LIN {X 0,Y 349.295,Z 384.118,A -85,B 0,C 180,E1 -15532.689,E2 -15532.689} C_VEL
LIN {X 0,Y 344.629,Z 399.806,A -85,B 0,C 180,E1 -15533.924,E2 -15533.924} C_VEL
LIN {X 0,Y 339.086,Z 417.351,A -85,B 0,C 180,E1 -15535.611,E2 -15535.611} C_VEL
LIN {X 0,Y 333.971,Z 433.133,A -85,B 0,C 180,E1 -15537.457,E2 -15537.457} C_VEL
LIN {X 0,Y 329.124,Z 447.831,A -85,B 0,C 180,E1 -15539.525,E2 -15539.525} C_VEL
LIN {X 0,Y 324.634,Z 461.889,A -85,B 0,C 180,E1 -15541.909,E2 -15541.909} C_VEL
LIN {X 0,Y 320.374,Z 475.464,A -85,B 0,C 180,E1 -15544.673,E2 -15544.673} C_VEL
LIN {X 0,Y 317.065,Z 486.958,A -85,B 0,C 180,E1 -15547.519,E2 -15547.519} C_VEL
LIN {X 0,Y 314.518,Z 496.621,A -85,B 0,C 180,E1 -15550.416,E2 -15550.416} C_VEL
LIN {X 0,Y 312.895,Z 503.797,A -85,B 0,C 180,E1 -15553.022,E2 -15553.022} C_VEL
LIN {X 0,Y 311.835,Z 509.983,A -85,B 0,C 180,E1 -15555.722,E2 -15555.722} C_VEL
LIN {X 0,Y 311.142,Z 514.648,A -85,B 0,C 180,E1 -15558.27,E2 -15558.27} C_VEL
LIN {X 0,Y 310.892,Z 518.384,A -85,B 0,C 180,E1 -15560.894,E2 -15560.894} C_VEL
LIN {X 0,Y 310.985,Z 521.013,A -85,B 0,C 180,E1 -15563.511,E2 -15563.511} C_VEL
LIN {X 0,Y 310.999,Z 522.524,A -85,B 0,C 180,E1 -15566.112,E2 -15566.112} C_VEL
LIN {X 0,Y 311.174,Z 522.908,A -85,B 0,C 180,E1 -15567.41,E2 -15567.41} C_VEL
LIN {X 0,Y 311.35,Z 522.705,A -85,B 0,C 180,E1 -15569.999,E2 -15569.999} C_VEL
LIN {X 0,Y 311.281,Z 521.372,A -85,B 0,C 180,E1 -15572.587,E2 -15572.587} C_VEL
LIN {X 0,Y 311.146,Z 518.832,A -85,B 0,C 180,E1 -15575.183,E2 -15575.183} C_VEL
LIN {X 0,Y 311.178,Z 516.141,A -85,B 0,C 180,E1 -15577.134,E2 -15577.134} C_VEL
LIN {X 0,Y 311.09,Z 511.33,A -85,B 0,C 180,E1 -15579.754,E2 -15579.754} C_VEL
LIN {X 0,Y 311.378,Z 505.192,A -85,B 0,C 180,E1 -15582.381,E2 -15582.381} C_VEL
LIN {X 0,Y 311.923,Z 497.582,A -85,B 0,C 180,E1 -15585.016,E2 -15585.016} C_VEL
LIN {X 0,Y 312.908,Z 488.328,A -85,B 0,C 180,E1 -15587.65,E2 -15587.65} C_VEL
LIN {X 0,Y 314.056,Z 478.588,A -85,B 0,C 180,E1 -15589.969,E2 -15589.969} C_VEL
LIN {X 0,Y 315.698,Z 467.285,A -85,B 0,C 180,E1 -15592.237,E2 -15592.237} C_VEL
LIN {X 0,Y 317.471,Z 454.864,A -85,B 0,C 180,E1 -15594.349,E2 -15594.349} C_VEL
LIN {X 0,Y 319.434,Z 441.443,A -85,B 0,C 180,E1 -15596.28,E2 -15596.28} C_VEL
LIN {X 0,Y 321.67,Z 427.047,A -85,B 0,C 180,E1 -15598.017,E2 -15598.017} C_VEL
LIN {X 0,Y 323.604,Z 413.175,A -85,B 0,C 180,E1 -15599.429,E2 -15599.429} C_VEL
LIN {X 0,Y 325.822,Z 396.562,A -85,B 0,C 180,E1 -15600.815,E2 -15600.815} C_VEL
LIN {X 0,Y 327.852,Z 379.404,A -85,B 0,C 180,E1 -15601.951,E2 -15601.951} C_VEL
LIN {X 0,Y 329.659,Z 361.75,A -85,B 0,C 180,E1 -15602.839,E2 -15602.839} C_VEL
LIN {X 0,Y 330.906,Z 344.404,A -85,B 0,C 180,E1 -15603.472,E2 -15603.472} C_VEL
LIN {X 0,Y 339.444,Z 199.123,A -85,B 0,C 180,E1 -15607.77,E2 -15607.77} C_VEL
LIN {X 0,Y 337.215,Z 179.474,A -85,B 0,C 180,E1 -15608.653,E2 -15608.653} C_VEL
LIN {X 0,Y 322.802,Z 147.216,A -85,B 0,C 180,E1 -15611.25,E2 -15611.25} C_VEL
LIN {X 0,Y 320.937,Z 143.018,A -85,B 0,C 180,E1 -15611.632,E2 -15611.632} C_VEL
LIN {X 0,Y 315.137,Z 125.785,A -85,B 0,C 180,E1 -15614.923,E2 -15614.923} C_VEL
LIN {X 0,Y 312.533,Z 117.869,A -85,B 0,C 180,E1 -15616.557,E2 -15616.557} C_VEL
LIN {X 0,Y 312.504,Z 117.869,A -85,B 0,C 180,E1 -15620.972,E2 -15620.972} C_VEL
LIN {X 0,Y 312.528,Z 117.87,A -85,B 0,C 180,E1 -15624.22,E2 -15624.22} C_VEL
LIN {X 0,Y 312.503,Z 117.868,A -85,B 0,C 180,E1 -15627.334,E2 -15627.334} C_VEL
LIN {X 0,Y 312.548,Z 117.863,A -85,B 0,C 180,E1 -15631.276,E2 -15631.276} C_VEL
LIN {X 0,Y 312.581,Z 117.86,A -85,B 0,C 180,E1 -15634.711,E2 -15634.711} C_VEL
LIN {X 0,Y 312.582,Z 117.86,A -85,B 0,C 180,E1 -15637.529,E2 -15637.529} C_VEL
LIN {X 0,Y 312.634,Z 117.855,A -85,B 0,C 180,E1 -15641.656,E2 -15641.656} C_VEL
LIN {X 0,Y 312.69,Z 117.848,A -85,B 0,C 180,E1 -15645.686,E2 -15645.686} C_VEL
LIN {X 0,Y 312.699,Z 117.846,A -85,B 0,C 180,E1 -15649.642,E2 -15649.642} C_VEL
LIN {X 0,Y 312.867,Z 117.824,A -85,B 0,C 180,E1 -15652.254,E2 -15652.254} C_VEL
LIN {X 0,Y 312.714,Z 117.839,A -85,B 0,C 180,E1 -15654.842,E2 -15654.842} C_VEL
LIN {X 0,Y 312.986,Z 117.808,A -85,B 0,C 180,E1 -15658.713,E2 -15658.713} C_VEL
LIN {X 0,Y 313.116,Z 117.794,A -85,B 0,C 180,E1 -15660,E2 -15660} C_VEL
LIN {X 0,Y 312.934,Z 117.814,A -85,B 0,C 180,E1 -15662.575,E2 -15662.575} C_VEL
LIN {X 0,Y 312.89,Z 117.818,A -85,B 0,C 180,E1 -15666.639,E2 -15666.639} C_VEL
LIN {X 0,Y 312.783,Z 117.835,A -85,B 0,C 180,E1 -15669.049,E2 -15669.049} C_VEL
LIN {X 0,Y 312.63,Z 117.853,A -85,B 0,C 180,E1 -15672.991,E2 -15672.991} C_VEL
LIN {X 0,Y 312.634,Z 117.854,A -85,B 0,C 180,E1 -15675.65,E2 -15675.65} C_VEL
LIN {X 0,Y 312.626,Z 117.857,A -85,B 0,C 180,E1 -15679.237,E2 -15679.237} C_VEL
LIN {X 0,Y 312.542,Z 117.864,A -85,B 0,C 180,E1 -15682.79,E2 -15682.79} C_VEL
LIN {X 0,Y 312.592,Z 117.857,A -85,B 0,C 180,E1 -15685.934,E2 -15685.934} C_VEL
LIN {X 0,Y 312.534,Z 117.864,A -85,B 0,C 180,E1 -15689.651,E2 -15689.651} C_VEL
LIN {X 0,Y 312.515,Z 117.867,A -85,B 0,C 180,E1 -15693.689,E2 -15693.689} C_VEL
LIN {X 0,Y 312.517,Z 117.867,A -85,B 0,C 180,E1 -15697.386,E2 -15697.386} C_VEL
LIN {X 0,Y 312.486,Z 117.873,A -85,B 0,C 180,E1 -15700.71,E2 -15700.71} C_VEL
LIN {X 0,Y 312.472,Z 117.872,A -85,B 0,C 180,E1 -15704.206,E2 -15704.206} C_VEL
LIN {X 0,Y 312.529,Z 117.864,A -85,B 0,C 180,E1 -15707.91,E2 -15707.91} C_VEL
LIN {X 0,Y 312.54,Z 117.863,A -85,B 0,C 180,E1 -15711.909,E2 -15711.909} C_VEL
LIN {X 0,Y 312.504,Z 117.867,A -85,B 0,C 180,E1 -15715.791,E2 -15715.791} C_VEL
LIN {X 0,Y 312.518,Z 117.869,A -85,B 0,C 180,E1 -15718.854,E2 -15718.854} C_VEL
LIN {X 0,Y 312.568,Z 117.858,A -85,B 0,C 180,E1 -15721.825,E2 -15721.825} C_VEL
LIN {X 0,Y 312.584,Z 117.861,A -85,B 0,C 180,E1 -15724.712,E2 -15724.712} C_VEL
LIN {X 0,Y 312.587,Z 117.857,A -85,B 0,C 180,E1 -15727.53,E2 -15727.53} C_VEL
LIN {X 0,Y 312.638,Z 117.851,A -85,B 0,C 180,E1 -15731.657,E2 -15731.657} C_VEL
LIN {X 0,Y 312.693,Z 117.844,A -85,B 0,C 180,E1 -15735.687,E2 -15735.687} C_VEL
LIN {X 0,Y 312.702,Z 117.844,A -85,B 0,C 180,E1 -15739.643,E2 -15739.643} C_VEL
LIN {X 0,Y 312.872,Z 117.827,A -85,B 0,C 180,E1 -15742.255,E2 -15742.255} C_VEL
LIN {X 0,Y 312.718,Z 117.841,A -85,B 0,C 180,E1 -15744.843,E2 -15744.843} C_VEL
LIN {X 0,Y 312.989,Z 117.808,A -85,B 0,C 180,E1 -15748.714,E2 -15748.714} C_VEL
LIN {X 0,Y 312.989,Z 117.807,A -85,B 0,C 180,E1 -15751.288,E2 -15751.288} C_VEL
LIN {X 0,Y 312.718,Z 117.84,A -85,B 0,C 180,E1 -15755.158,E2 -15755.158} C_VEL
LIN {X 0,Y 312.873,Z 117.826,A -85,B 0,C 180,E1 -15757.747,E2 -15757.747} C_VEL
LIN {X 0,Y 312.671,Z 117.849,A -85,B 0,C 180,E1 -15761.672,E2 -15761.672} C_VEL
LIN {X 0,Y 312.702,Z 117.844,A -85,B 0,C 180,E1 -15764.888,E2 -15764.888} C_VEL
LIN {X 0,Y 312.632,Z 117.852,A -85,B 0,C 180,E1 -15769.237,E2 -15769.237} C_VEL
LIN {X 0,Y 312.548,Z 117.861,A -85,B 0,C 180,E1 -15772.79,E2 -15772.79} C_VEL
LIN {X 0,Y 312.605,Z 117.858,A -85,B 0,C 180,E1 -15775.936,E2 -15775.936} C_VEL
LIN {X 0,Y 312.54,Z 117.868,A -85,B 0,C 180,E1 -15779.651,E2 -15779.651} C_VEL
LIN {X 0,Y 312.522,Z 117.869,A -85,B 0,C 180,E1 -15783.689,E2 -15783.689} C_VEL
LIN {X 0,Y 312.541,Z 117.868,A -85,B 0,C 180,E1 -15787.384,E2 -15787.384} C_VEL
LIN {X 0,Y 312.493,Z 117.869,A -85,B 0,C 180,E1 -15790.71,E2 -15790.71} C_VEL
LIN {X 0,Y 312.476,Z 117.872,A -85,B 0,C 180,E1 -15794.206,E2 -15794.206} C_VEL
LIN {X 0,Y 312.489,Z 117.872,A -85,B 0,C 180,E1 -15797.919,E2 -15797.919} C_VEL
LIN {X 0,Y 312.489,Z 117.887,A -85,B 0,C 180,E1 -15798.632,E2 -15798.632} C_VEL
LIN {X 0,Y 313.513,Z 120.747,A -85,B 0,C 180,E1 -15798.857,E2 -15798.857} C_VEL
LIN {X 0,Y 325.494,Z 143.603,A -85,B 0,C 180,E1 -15800.977,E2 -15800.977} C_VEL
LIN {X 0,Y 338.412,Z 169.69,A -85,B 0,C 180,E1 -15803.121,E2 -15803.121} C_VEL
LIN {X 0,Y 336.711,Z 199.183,A -85,B 0,C 180,E1 -15803.99,E2 -15803.99} C_VEL
LIN {X 0,Y 331.473,Z 290.627,A -85,B 0,C 180,E1 -15806.67,E2 -15806.67} C_VEL
LIN {X 0,Y 330.453,Z 296.401,A -85,B 0,C 180,E1 -15806.798,E2 -15806.798} C_VEL
LIN {X 0,Y 323.959,Z 315.007,A -85,B 0,C 180,E1 -15807.144,E2 -15807.144} C_VEL
LIN {X 0,Y 322.988,Z 320.671,A -85,B 0,C 180,E1 -15807.384,E2 -15807.384} C_VEL
LIN {X 0,Y 321.504,Z 337.305,A -85,B 0,C 180,E1 -15808.356,E2 -15808.356} C_VEL
LIN {X 0,Y 319.895,Z 352.792,A -85,B 0,C 180,E1 -15809.495,E2 -15809.495} C_VEL
LIN {X 0,Y 318.015,Z 368.566,A -85,B 0,C 180,E1 -15810.909,E2 -15810.909} C_VEL
LIN {X 0,Y 315.817,Z 384.138,A -85,B 0,C 180,E1 -15812.592,E2 -15812.592} C_VEL
LIN {X 0,Y 313.777,Z 398.504,A -85,B 0,C 180,E1 -15814.459,E2 -15814.459} C_VEL
LIN {X 0,Y 311.835,Z 411.307,A -85,B 0,C 180,E1 -15816.419,E2 -15816.419} C_VEL
LIN {X 0,Y 309.955,Z 424.018,A -85,B 0,C 180,E1 -15818.728,E2 -15818.728} C_VEL
LIN {X 0,Y 308.326,Z 434.772,A -85,B 0,C 180,E1 -15821.046,E2 -15821.046} C_VEL
LIN {X 0,Y 307.039,Z 443.961,A -85,B 0,C 180,E1 -15823.374,E2 -15823.374} C_VEL
LIN {X 0,Y 305.92,Z 452.844,A -85,B 0,C 180,E1 -15826.041,E2 -15826.041} C_VEL
LIN {X 0,Y 305.072,Z 460.203,A -85,B 0,C 180,E1 -15828.707,E2 -15828.707} C_VEL
LIN {X 0,Y 304.599,Z 466.158,A -85,B 0,C 180,E1 -15831.374,E2 -15831.374} C_VEL
LIN {X 0,Y 304.269,Z 470.833,A -85,B 0,C 180,E1 -15834.034,E2 -15834.034} C_VEL
LIN {X 0,Y 304.16,Z 473.616,A -85,B 0,C 180,E1 -15836.025,E2 -15836.025} C_VEL
LIN {X 0,Y 304.172,Z 476.328,A -85,B 0,C 180,E1 -15838.676,E2 -15838.676} C_VEL
LIN {X 0,Y 304.288,Z 478.039,A -85,B 0,C 180,E1 -15841.323,E2 -15841.323} C_VEL
LIN {X 0,Y 304.671,Z 478.631,A -85,B 0,C 180,E1 -15843.968,E2 -15843.968} C_VEL
LIN {X 0,Y 305.028,Z 478.313,A -85,B 0,C 180,E1 -15846.615,E2 -15846.615} C_VEL
LIN {X 0,Y 305.938,Z 476.894,A -85,B 0,C 180,E1 -15849.253,E2 -15849.253} C_VEL
LIN {X 0,Y 307.056,Z 474.523,A -85,B 0,C 180,E1 -15851.888,E2 -15851.888} C_VEL
LIN {X 0,Y 308.567,Z 471.116,A -85,B 0,C 180,E1 -15854.509,E2 -15854.509} C_VEL
LIN {X 0,Y 310.423,Z 466.643,A -85,B 0,C 180,E1 -15857.117,E2 -15857.117} C_VEL
LIN {X 0,Y 312.955,Z 461.065,A -85,B 0,C 180,E1 -15859.685,E2 -15859.685} C_VEL
LIN {X 0,Y 315.894,Z 454.246,A -85,B 0,C 180,E1 -15862.223,E2 -15862.223} C_VEL
LIN {X 0,Y 319.439,Z 446.086,A -85,B 0,C 180,E1 -15864.709,E2 -15864.709} C_VEL
LIN {X 0,Y 323.477,Z 436.53,A -85,B 0,C 180,E1 -15867.145,E2 -15867.145} C_VEL
LIN {X 0,Y 328.04,Z 425.33,A -85,B 0,C 180,E1 -15869.522,E2 -15869.522} C_VEL
LIN {X 0,Y 333.3,Z 412.161,A -85,B 0,C 180,E1 -15871.813,E2 -15871.813} C_VEL
LIN {X 0,Y 338.512,Z 398.159,A -85,B 0,C 180,E1 -15873.853,E2 -15873.853} C_VEL
LIN {X 0,Y 343.392,Z 384.43,A -85,B 0,C 180,E1 -15875.502,E2 -15875.502} C_VEL
LIN {X 0,Y 348.987,Z 367.579,A -85,B 0,C 180,E1 -15877.167,E2 -15877.167} C_VEL
LIN {X 0,Y 354.438,Z 349.416,A -85,B 0,C 180,E1 -15878.611,E2 -15878.611} C_VEL
LIN {X 0,Y 358.655,Z 333.375,A -85,B 0,C 180,E1 -15879.625,E2 -15879.625} C_VEL
LIN {X 0,Y 362.306,Z 317.392,A -85,B 0,C 180,E1 -15880.415,E2 -15880.415} C_VEL
LIN {X 0,Y 369.736,Z 283.735,A -85,B 0,C 180,E1 -15881.704,E2 -15881.704} C_VEL
LIN {X 0,Y 385.229,Z 220.867,A -85,B 0,C 180,E1 -15883.972,E2 -15883.972} C_VEL
LIN {X 0,Y 386.116,Z 217.532,A -85,B 0,C 180,E1 -15884.081,E2 -15884.081} C_VEL
LIN {X 0,Y 385.94,Z 218.526,A -85,B 0,C 180,E1 -15884.797,E2 -15884.797} C_VEL
LIN {X 0,Y 369.925,Z 285.407,A -85,B 0,C 180,E1 -15887.172,E2 -15887.172} C_VEL
LIN {X 0,Y 357.945,Z 341.127,A -85,B 0,C 180,E1 -15889.289,E2 -15889.289} C_VEL
LIN {X 0,Y 352.257,Z 362.801,A -85,B 0,C 180,E1 -15890.323,E2 -15890.323} C_VEL
LIN {X 0,Y 346.181,Z 382.739,A -85,B 0,C 180,E1 -15891.556,E2 -15891.556} C_VEL
LIN {X 0,Y 341.651,Z 396.692,A -85,B 0,C 180,E1 -15892.638,E2 -15892.638} C_VEL
LIN {X 0,Y 335.68,Z 414.246,A -85,B 0,C 180,E1 -15894.294,E2 -15894.294} C_VEL
LIN {X 0,Y 330.21,Z 429.88,A -85,B 0,C 180,E1 -15896.104,E2 -15896.104} C_VEL
LIN {X 0,Y 325.165,Z 443.856,A -85,B 0,C 180,E1 -15898.025,E2 -15898.025} C_VEL
LIN {X 0,Y 320.164,Z 458.156,A -85,B 0,C 180,E1 -15900.402,E2 -15900.402} C_VEL
LIN {X 0,Y 315.91,Z 470.554,A -85,B 0,C 180,E1 -15902.857,E2 -15902.857} C_VEL
LIN {X 0,Y 312.361,Z 481.394,A -85,B 0,C 180,E1 -15905.402,E2 -15905.402} C_VEL
LIN {X 0,Y 309.46,Z 490.728,A -85,B 0,C 180,E1 -15907.992,E2 -15907.992} C_VEL
LIN {X 0,Y 307.28,Z 498.66,A -85,B 0,C 180,E1 -15910.631,E2 -15910.631} C_VEL
LIN {X 0,Y 305.658,Z 505.427,A -85,B 0,C 180,E1 -15913.296,E2 -15913.296} C_VEL
LIN {X 0,Y 304.618,Z 511.205,A -85,B 0,C 180,E1 -15916.109,E2 -15916.109} C_VEL
LIN {X 0,Y 304.111,Z 514.415,A -85,B 0,C 180,E1 -15917.995,E2 -15917.995} C_VEL
LIN {X 0,Y 303.814,Z 517.998,A -85,B 0,C 180,E1 -15920.68,E2 -15920.68} C_VEL
LIN {X 0,Y 303.901,Z 520.568,A -85,B 0,C 180,E1 -15923.359,E2 -15923.359} C_VEL
LIN {X 0,Y 303.924,Z 521.949,A -85,B 0,C 180,E1 -15926.021,E2 -15926.021} C_VEL
LIN {X 0,Y 304.173,Z 522.312,A -85,B 0,C 180,E1 -15928.675,E2 -15928.675} C_VEL
LIN {X 0,Y 304.296,Z 522.014,A -85,B 0,C 180,E1 -15929.999,E2 -15929.999} C_VEL
LIN {X 0,Y 304.222,Z 520.551,A -85,B 0,C 180,E1 -15932.647,E2 -15932.647} C_VEL
LIN {X 0,Y 304.095,Z 517.939,A -85,B 0,C 180,E1 -15935.303,E2 -15935.303} C_VEL
LIN {X 0,Y 304.12,Z 515.109,A -85,B 0,C 180,E1 -15937.301,E2 -15937.301} C_VEL
LIN {X 0,Y 304.051,Z 510.224,A -85,B 0,C 180,E1 -15939.982,E2 -15939.982} C_VEL
LIN {X 0,Y 304.354,Z 503.921,A -85,B 0,C 180,E1 -15942.671,E2 -15942.671} C_VEL
LIN {X 0,Y 304.966,Z 496.129,A -85,B 0,C 180,E1 -15945.367,E2 -15945.367} C_VEL
LIN {X 0,Y 305.961,Z 486.65,A -85,B 0,C 180,E1 -15948.064,E2 -15948.064} C_VEL
LIN {X 0,Y 307.187,Z 476.958,A -85,B 0,C 180,E1 -15950.384,E2 -15950.384} C_VEL
LIN {X 0,Y 308.889,Z 465.211,A -85,B 0,C 180,E1 -15952.754,E2 -15952.754} C_VEL
LIN {X 0,Y 310.981,Z 451.483,A -85,B 0,C 180,E1 -15955.07,E2 -15955.07} C_VEL
LIN {X 0,Y 313.084,Z 437.545,A -85,B 0,C 180,E1 -15957.036,E2 -15957.036} C_VEL
LIN {X 0,Y 315.198,Z 423.926,A -85,B 0,C 180,E1 -15958.644,E2 -15958.644} C_VEL
LIN {X 0,Y 317.431,Z 408.668,A -85,B 0,C 180,E1 -15960.155,E2 -15960.155} C_VEL
LIN {X 0,Y 319.559,Z 392.24,A -85,B 0,C 180,E1 -15961.488,E2 -15961.488} C_VEL
LIN {X 0,Y 321.572,Z 375.515,A -85,B 0,C 180,E1 -15962.559,E2 -15962.559} C_VEL
LIN {X 0,Y 323.267,Z 358.638,A -85,B 0,C 180,E1 -15963.387,E2 -15963.387} C_VEL
LIN {X 0,Y 324.53,Z 340.629,A -85,B 0,C 180,E1 -15964.032,E2 -15964.032} C_VEL
LIN {X 0,Y 333.127,Z 199.897,A -85,B 0,C 180,E1 -15968.302,E2 -15968.302} C_VEL
LIN {X 0,Y 331.193,Z 182.224,A -85,B 0,C 180,E1 -15969.12,E2 -15969.12} C_VEL
LIN {X 0,Y 316.998,Z 150.393,A -85,B 0,C 180,E1 -15971.74,E2 -15971.74} C_VEL
LIN {X 0,Y 313.451,Z 142.568,A -85,B 0,C 180,E1 -15972.449,E2 -15972.449} C_VEL
LIN {X 0,Y 308.276,Z 127.199,A -85,B 0,C 180,E1 -15975.464,E2 -15975.464} C_VEL
LIN {X 0,Y 305.451,Z 118.749,A -85,B 0,C 180,E1 -15977.231,E2 -15977.231} C_VEL
LIN {X 0,Y 305.454,Z 118.75,A -85,B 0,C 180,E1 -15979.892,E2 -15979.892} C_VEL
LIN {X 0,Y 305.495,Z 118.742,A -85,B 0,C 180,E1 -15983.626,E2 -15983.626} C_VEL
LIN {X 0,Y 305.461,Z 118.749,A -85,B 0,C 180,E1 -15986.483,E2 -15986.483} C_VEL
LIN {X 0,Y 305.462,Z 118.747,A -85,B 0,C 180,E1 -15989.591,E2 -15989.591} C_VEL
LIN {X 0,Y 305.517,Z 118.741,A -85,B 0,C 180,E1 -15992.608,E2 -15992.608} C_VEL
LIN {X 0,Y 305.503,Z 118.743,A -85,B 0,C 180,E1 -15995.539,E2 -15995.539} C_VEL
LIN {X 0,Y 305.515,Z 118.743,A -85,B 0,C 180,E1 -15999.815,E2 -15999.815} C_VEL
LIN {X 0,Y 305.57,Z 118.731,A -85,B 0,C 180,E1 -16002.603,E2 -16002.603} C_VEL
LIN {X 0,Y 305.644,Z 118.724,A -85,B 0,C 180,E1 -16005.349,E2 -16005.349} C_VEL
LIN {X 0,Y 305.636,Z 118.724,A -85,B 0,C 180,E1 -16009.4,E2 -16009.4} C_VEL
LIN {X 0,Y 305.808,Z 118.704,A -85,B 0,C 180,E1 -16012.074,E2 -16012.074} C_VEL
LIN {X 0,Y 305.685,Z 118.714,A -85,B 0,C 180,E1 -16014.724,E2 -16014.724} C_VEL
LIN {X 0,Y 305.953,Z 118.684,A -85,B 0,C 180,E1 -16018.684,E2 -16018.684} C_VEL
LIN {X 0,Y 305.953,Z 118.686,A -85,B 0,C 180,E1 -16021.316,E2 -16021.316} C_VEL
LIN {X 0,Y 305.848,Z 118.696,A -85,B 0,C 180,E1 -16026.598,E2 -16026.598} C_VEL
LIN {X 0,Y 305.731,Z 118.715,A -85,B 0,C 180,E1 -16029.26,E2 -16029.26} C_VEL
LIN {X 0,Y 305.585,Z 118.733,A -85,B 0,C 180,E1 -16033.296,E2 -16033.296} C_VEL
LIN {X 0,Y 305.589,Z 118.729,A -85,B 0,C 180,E1 -16036.02,E2 -16036.02} C_VEL
LIN {X 0,Y 305.572,Z 118.735,A -85,B 0,C 180,E1 -16039.445,E2 -16039.445} C_VEL
LIN {X 0,Y 305.487,Z 118.745,A -85,B 0,C 180,E1 -16043.042,E2 -16043.042} C_VEL
LIN {X 0,Y 305.521,Z 118.737,A -85,B 0,C 180,E1 -16046.219,E2 -16046.219} C_VEL
LIN {X 0,Y 305.484,Z 118.747,A -85,B 0,C 180,E1 -16049.048,E2 -16049.048} C_VEL
LIN {X 0,Y 305.438,Z 118.747,A -85,B 0,C 180,E1 -16051.953,E2 -16051.953} C_VEL
LIN {X 0,Y 305.459,Z 118.75,A -85,B 0,C 180,E1 -16055.114,E2 -16055.114} C_VEL
LIN {X 0,Y 305.437,Z 118.748,A -85,B 0,C 180,E1 -16058.527,E2 -16058.527} C_VEL
LIN {X 0,Y 305.456,Z 118.748,A -85,B 0,C 180,E1 -16062.587,E2 -16062.587} C_VEL
LIN {X 0,Y 305.476,Z 118.743,A -85,B 0,C 180,E1 -16066.355,E2 -16066.355} C_VEL
LIN {X 0,Y 305.462,Z 118.745,A -85,B 0,C 180,E1 -16069.894,E2 -16069.894} C_VEL
LIN {X 0,Y 305.497,Z 118.739,A -85,B 0,C 180,E1 -16073.628,E2 -16073.628} C_VEL
LIN {X 0,Y 305.463,Z 118.748,A -85,B 0,C 180,E1 -16076.484,E2 -16076.484} C_VEL
LIN {X 0,Y 305.455,Z 118.745,A -85,B 0,C 180,E1 -16079.591,E2 -16079.591} C_VEL
LIN {X 0,Y 305.513,Z 118.743,A -85,B 0,C 180,E1 -16082.609,E2 -16082.609} C_VEL
LIN {X 0,Y 305.507,Z 118.739,A -85,B 0,C 180,E1 -16085.54,E2 -16085.54} C_VEL
LIN {X 0,Y 305.529,Z 118.736,A -85,B 0,C 180,E1 -16089.817,E2 -16089.817} C_VEL
LIN {X 0,Y 305.574,Z 118.734,A -85,B 0,C 180,E1 -16092.604,E2 -16092.604} C_VEL
LIN {X 0,Y 305.648,Z 118.72,A -85,B 0,C 180,E1 -16095.35,E2 -16095.35} C_VEL
LIN {X 0,Y 305.639,Z 118.723,A -85,B 0,C 180,E1 -16099.401,E2 -16099.401} C_VEL
LIN {X 0,Y 305.813,Z 118.704,A -85,B 0,C 180,E1 -16102.075,E2 -16102.075} C_VEL
LIN {X 0,Y 305.689,Z 118.718,A -85,B 0,C 180,E1 -16104.724,E2 -16104.724} C_VEL
LIN {X 0,Y 305.956,Z 118.684,A -85,B 0,C 180,E1 -16108.685,E2 -16108.685} C_VEL
LIN {X 0,Y 305.956,Z 118.683,A -85,B 0,C 180,E1 -16111.317,E2 -16111.317} C_VEL
LIN {X 0,Y 305.854,Z 118.697,A -85,B 0,C 180,E1 -16116.598,E2 -16116.598} C_VEL
LIN {X 0,Y 305.737,Z 118.712,A -85,B 0,C 180,E1 -16119.261,E2 -16119.261} C_VEL
LIN {X 0,Y 305.59,Z 118.73,A -85,B 0,C 180,E1 -16123.297,E2 -16123.297} C_VEL
LIN {X 0,Y 305.596,Z 118.731,A -85,B 0,C 180,E1 -16126.021,E2 -16126.021} C_VEL
LIN {X 0,Y 305.578,Z 118.732,A -85,B 0,C 180,E1 -16129.445,E2 -16129.445} C_VEL
LIN {X 0,Y 305.493,Z 118.741,A -85,B 0,C 180,E1 -16133.042,E2 -16133.042} C_VEL
LIN {X 0,Y 305.534,Z 118.737,A -85,B 0,C 180,E1 -16136.222,E2 -16136.222} C_VEL
LIN {X 0,Y 305.49,Z 118.743,A -85,B 0,C 180,E1 -16139.048,E2 -16139.048} C_VEL
LIN {X 0,Y 305.445,Z 118.75,A -85,B 0,C 180,E1 -16141.953,E2 -16141.953} C_VEL
LIN {X 0,Y 305.466,Z 118.747,A -85,B 0,C 180,E1 -16145.114,E2 -16145.114} C_VEL
LIN {X 0,Y 305.47,Z 118.745,A -85,B 0,C 180,E1 -16148.534,E2 -16148.534} C_VEL
LIN {X 0,Y 305.462,Z 118.746,A -85,B 0,C 180,E1 -16152.587,E2 -16152.587} C_VEL
LIN {X 0,Y 305.446,Z 118.749,A -85,B 0,C 180,E1 -16156.349,E2 -16156.349} C_VEL
LIN {X 0,Y 305.444,Z 118.75,A -85,B 0,C 180,E1 -16157.881,E2 -16157.881} C_VEL
LIN {X 0,Y 306.47,Z 121.618,A -85,B 0,C 180,E1 -16158.117,E2 -16158.117} C_VEL
LIN {X 0,Y 317.846,Z 143.327,A -85,B 0,C 180,E1 -16160.2,E2 -16160.2} C_VEL
LIN {X 0,Y 330.366,Z 168.475,A -85,B 0,C 180,E1 -16162.352,E2 -16162.352} C_VEL
LIN {X 0,Y 332.116,Z 171.994,A -85,B 0,C 180,E1 -16162.637,E2 -16162.637} C_VEL
LIN {X 0,Y 324.12,Z 304.568,A -85,B 0,C 180,E1 -16166.665,E2 -16166.665} C_VEL
LIN {X 0,Y 322.988,Z 320.671,A -85,B 0,C 180,E1 -16167.384,E2 -16167.384} C_VEL
LIN {X 0,Y 321.887,Z 326.318,A -85,B 0,C 180,E1 -16167.633,E2 -16167.633} C_VEL
LIN {X 0,Y 315.296,Z 342.492,A -85,B 0,C 180,E1 -16168.33,E2 -16168.33} C_VEL
LIN {X 0,Y 313.78,Z 347.884,A -85,B 0,C 180,E1 -16168.675,E2 -16168.675} C_VEL
LIN {X 0,Y 313.531,Z 349.686,A -85,B 0,C 180,E1 -16168.813,E2 -16168.813} C_VEL
LIN {X 0,Y 311.592,Z 366.064,A -85,B 0,C 180,E1 -16170.25,E2 -16170.25} C_VEL
LIN {X 0,Y 309.442,Z 381.708,A -85,B 0,C 180,E1 -16171.918,E2 -16171.918} C_VEL
LIN {X 0,Y 307.178,Z 396.902,A -85,B 0,C 180,E1 -16173.869,E2 -16173.869} C_VEL
LIN {X 0,Y 305.006,Z 410.994,A -85,B 0,C 180,E1 -16176.039,E2 -16176.039} C_VEL
LIN {X 0,Y 303.174,Z 422.953,A -85,B 0,C 180,E1 -16178.229,E2 -16178.229} C_VEL
LIN {X 0,Y 301.491,Z 433.971,A -85,B 0,C 180,E1 -16180.599,E2 -16180.599} C_VEL
LIN {X 0,Y 299.94,Z 444.616,A -85,B 0,C 180,E1 -16183.319,E2 -16183.319} C_VEL
LIN {X 0,Y 298.927,Z 452.498,A -85,B 0,C 180,E1 -16185.708,E2 -16185.708} C_VEL
LIN {X 0,Y 298.057,Z 460.036,A -85,B 0,C 180,E1 -16188.438,E2 -16188.438} C_VEL
LIN {X 0,Y 297.541,Z 466.123,A -85,B 0,C 180,E1 -16191.168,E2 -16191.168} C_VEL
LIN {X 0,Y 297.224,Z 470.638,A -85,B 0,C 180,E1 -16193.671,E2 -16193.671} C_VEL
LIN {X 0,Y 297.084,Z 473.84,A -85,B 0,C 180,E1 -16195.93,E2 -16195.93} C_VEL
LIN {X 0,Y 297.097,Z 476.723,A -85,B 0,C 180,E1 -16198.644,E2 -16198.644} C_VEL
LIN {X 0,Y 297.23,Z 478.522,A -85,B 0,C 180,E1 -16201.355,E2 -16201.355} C_VEL
LIN {X 0,Y 297.634,Z 479.285,A -85,B 0,C 180,E1 -16204.062,E2 -16204.062} C_VEL
LIN {X 0,Y 298.007,Z 479.102,A -85,B 0,C 180,E1 -16206.772,E2 -16206.772} C_VEL
LIN {X 0,Y 298.996,Z 477.823,A -85,B 0,C 180,E1 -16209.47,E2 -16209.47} C_VEL
LIN {X 0,Y 300.18,Z 475.644,A -85,B 0,C 180,E1 -16212.164,E2 -16212.164} C_VEL
LIN {X 0,Y 301.785,Z 472.359,A -85,B 0,C 180,E1 -16214.843,E2 -16214.843} C_VEL
LIN {X 0,Y 303.795,Z 468.104,A -85,B 0,C 180,E1 -16217.502,E2 -16217.502} C_VEL
LIN {X 0,Y 306.457,Z 462.717,A -85,B 0,C 180,E1 -16220.12,E2 -16220.12} C_VEL
LIN {X 0,Y 309.571,Z 456.139,A -85,B 0,C 180,E1 -16222.702,E2 -16222.702} C_VEL
LIN {X 0,Y 313.823,Z 447.22,A -85,B 0,C 180,E1 -16225.537,E2 -16225.537} C_VEL
LIN {X 0,Y 318.607,Z 436.807,A -85,B 0,C 180,E1 -16228.239,E2 -16228.239} C_VEL
LIN {X 0,Y 323.707,Z 425.368,A -85,B 0,C 180,E1 -16230.677,E2 -16230.677} C_VEL
LIN {X 0,Y 329.182,Z 412.692,A -85,B 0,C 180,E1 -16232.897,E2 -16232.897} C_VEL
LIN {X 0,Y 334.343,Z 399.984,A -85,B 0,C 180,E1 -16234.781,E2 -16234.781} C_VEL
LIN {X 0,Y 340.193,Z 384.903,A -85,B 0,C 180,E1 -16236.621,E2 -16236.621} C_VEL
LIN {X 0,Y 346.139,Z 368.406,A -85,B 0,C 180,E1 -16238.263,E2 -16238.263} C_VEL
LIN {X 0,Y 352.071,Z 350.278,A -85,B 0,C 180,E1 -16239.701,E2 -16239.701} C_VEL
LIN {X 0,Y 357.004,Z 332.93,A -85,B 0,C 180,E1 -16240.793,E2 -16240.793} C_VEL
LIN {X 0,Y 360.932,Z 317.028,A -85,B 0,C 180,E1 -16241.549,E2 -16241.549} C_VEL
LIN {X 0,Y 368.295,Z 285.984,A -85,B 0,C 180,E1 -16242.736,E2 -16242.736} C_VEL
LIN {X 0,Y 379.914,Z 240.914,A -85,B 0,C 180,E1 -16244.361,E2 -16244.361} C_VEL
LIN {X 0,Y 379.946,Z 240.817,A -85,B 0,C 180,E1 -16244.488,E2 -16244.488} C_VEL
LIN {X 0,Y 363.378,Z 308.568,A -85,B 0,C 180,E1 -16246.923,E2 -16246.923} C_VEL
LIN {X 0,Y 355.799,Z 341.181,A -85,B 0,C 180,E1 -16248.19,E2 -16248.19} C_VEL
LIN {X 0,Y 350.001,Z 361.561,A -85,B 0,C 180,E1 -16249.166,E2 -16249.166} C_VEL
LIN {X 0,Y 343.867,Z 380.336,A -85,B 0,C 180,E1 -16250.305,E2 -16250.305} C_VEL
LIN {X 0,Y 338.469,Z 395.611,A -85,B 0,C 180,E1 -16251.469,E2 -16251.469} C_VEL
LIN {X 0,Y 331.672,Z 414.098,A -85,B 0,C 180,E1 -16253.229,E2 -16253.229} C_VEL
LIN {X 0,Y 325.691,Z 429.802,A -85,B 0,C 180,E1 -16255.083,E2 -16255.083} C_VEL
LIN {X 0,Y 320.118,Z 444.005,A -85,B 0,C 180,E1 -16257.086,E2 -16257.086} C_VEL
LIN {X 0,Y 314.758,Z 458.002,A -85,B 0,C 180,E1 -16259.471,E2 -16259.471} C_VEL
LIN {X 0,Y 310.18,Z 470.185,A -85,B 0,C 180,E1 -16261.951,E2 -16261.951} C_VEL
LIN {X 0,Y 306.345,Z 480.85,A -85,B 0,C 180,E1 -16264.522,E2 -16264.522} C_VEL
LIN {X 0,Y 302.851,Z 491.14,A -85,B 0,C 180,E1 -16267.486,E2 -16267.486} C_VEL
LIN {X 0,Y 300.521,Z 498.875,A -85,B 0,C 180,E1 -16270.177,E2 -16270.177} C_VEL
LIN {X 0,Y 298.757,Z 505.411,A -85,B 0,C 180,E1 -16272.898,E2 -16272.898} C_VEL
LIN {X 0,Y 297.774,Z 510.37,A -85,B 0,C 180,E1 -16275.391,E2 -16275.391} C_VEL
LIN {X 0,Y 297.086,Z 514.186,A -85,B 0,C 180,E1 -16277.706,E2 -16277.706} C_VEL
LIN {X 0,Y 296.711,Z 517.629,A -85,B 0,C 180,E1 -16280.455,E2 -16280.455} C_VEL
LIN {X 0,Y 296.8,Z 520.084,A -85,B 0,C 180,E1 -16283.2,E2 -16283.2} C_VEL
LIN {X 0,Y 296.853,Z 521.378,A -85,B 0,C 180,E1 -16285.926,E2 -16285.926} C_VEL
LIN {X 0,Y 297.113,Z 521.607,A -85,B 0,C 180,E1 -16288.644,E2 -16288.644} C_VEL
LIN {X 0,Y 297.228,Z 521.312,A -85,B 0,C 180,E1 -16289.999,E2 -16289.999} C_VEL
LIN {X 0,Y 297.165,Z 519.712,A -85,B 0,C 180,E1 -16292.71,E2 -16292.71} C_VEL
LIN {X 0,Y 297.046,Z 516.967,A -85,B 0,C 180,E1 -16295.43,E2 -16295.43} C_VEL
LIN {X 0,Y 297.064,Z 514.055,A -85,B 0,C 180,E1 -16297.476,E2 -16297.476} C_VEL
LIN {X 0,Y 297.019,Z 509.045,A -85,B 0,C 180,E1 -16300.221,E2 -16300.221} C_VEL
LIN {X 0,Y 297.344,Z 502.603,A -85,B 0,C 180,E1 -16302.975,E2 -16302.975} C_VEL
LIN {X 0,Y 298.025,Z 494.619,A -85,B 0,C 180,E1 -16305.734,E2 -16305.734} C_VEL
LIN {X 0,Y 299.096,Z 484.925,A -85,B 0,C 180,E1 -16308.494,E2 -16308.494} C_VEL
LIN {X 0,Y 300.34,Z 474.809,A -85,B 0,C 180,E1 -16310.906,E2 -16310.906} C_VEL
LIN {X 0,Y 301.892,Z 464.828,A -85,B 0,C 180,E1 -16312.95,E2 -16312.95} C_VEL
LIN {X 0,Y 303.993,Z 451.404,A -85,B 0,C 180,E1 -16315.273,E2 -16315.273} C_VEL
LIN {X 0,Y 306.182,Z 437.216,A -85,B 0,C 180,E1 -16317.326,E2 -16317.326} C_VEL
LIN {X 0,Y 308.332,Z 423.639,A -85,B 0,C 180,E1 -16318.97,E2 -16318.97} C_VEL
LIN {X 0,Y 310.666,Z 407.829,A -85,B 0,C 180,E1 -16320.571,E2 -16320.571} C_VEL
LIN {X 0,Y 312.918,Z 391.067,A -85,B 0,C 180,E1 -16321.951,E2 -16321.951} C_VEL
LIN {X 0,Y 314.999,Z 374.259,A -85,B 0,C 180,E1 -16323.039,E2 -16323.039} C_VEL
LIN {X 0,Y 316.802,Z 356.286,A -85,B 0,C 180,E1 -16323.921,E2 -16323.921} C_VEL
LIN {X 0,Y 318.279,Z 333.979,A -85,B 0,C 180,E1 -16324.699,E2 -16324.699} C_VEL
LIN {X 0,Y 326.798,Z 200.494,A -85,B 0,C 180,E1 -16328.862,E2 -16328.862} C_VEL
LIN {X 0,Y 325.007,Z 184.648,A -85,B 0,C 180,E1 -16329.614,E2 -16329.614} C_VEL
LIN {X 0,Y 311.248,Z 153.667,A -85,B 0,C 180,E1 -16332.221,E2 -16332.221} C_VEL
LIN {X 0,Y 305.936,Z 142.033,A -85,B 0,C 180,E1 -16333.311,E2 -16333.311} C_VEL
LIN {X 0,Y 301.313,Z 128.379,A -85,B 0,C 180,E1 -16336.061,E2 -16336.061} C_VEL
LIN {X 0,Y 298.422,Z 119.627,A -85,B 0,C 180,E1 -16337.955,E2 -16337.955} C_VEL
LIN {X 0,Y 298.427,Z 119.627,A -85,B 0,C 180,E1 -16342.244,E2 -16342.244} C_VEL
LIN {X 0,Y 298.404,Z 119.626,A -85,B 0,C 180,E1 -16345.581,E2 -16345.581} C_VEL
LIN {X 0,Y 298.394,Z 119.627,A -85,B 0,C 180,E1 -16348.791,E2 -16348.791} C_VEL
LIN {X 0,Y 298.459,Z 119.622,A -85,B 0,C 180,E1 -16351.904,E2 -16351.904} C_VEL
LIN {X 0,Y 298.481,Z 119.617,A -85,B 0,C 180,E1 -16354.924,E2 -16354.924} C_VEL
LIN {X 0,Y 298.445,Z 119.62,A -85,B 0,C 180,E1 -16359.315,E2 -16359.315} C_VEL
LIN {X 0,Y 298.534,Z 119.61,A -85,B 0,C 180,E1 -16362.179,E2 -16362.179} C_VEL
LIN {X 0,Y 298.589,Z 119.602,A -85,B 0,C 180,E1 -16364.995,E2 -16364.995} C_VEL
LIN {X 0,Y 298.591,Z 119.6,A -85,B 0,C 180,E1 -16369.147,E2 -16369.147} C_VEL
LIN {X 0,Y 298.754,Z 119.585,A -85,B 0,C 180,E1 -16371.886,E2 -16371.886} C_VEL
LIN {X 0,Y 298.656,Z 119.589,A -85,B 0,C 180,E1 -16374.599,E2 -16374.599} C_VEL
LIN {X 0,Y 298.919,Z 119.56,A -85,B 0,C 180,E1 -16378.653,E2 -16378.653} C_VEL
LIN {X 0,Y 298.919,Z 119.563,A -85,B 0,C 180,E1 -16381.347,E2 -16381.347} C_VEL
LIN {X 0,Y 298.794,Z 119.575,A -85,B 0,C 180,E1 -16386.754,E2 -16386.754} C_VEL
LIN {X 0,Y 298.676,Z 119.595,A -85,B 0,C 180,E1 -16389.481,E2 -16389.481} C_VEL
LIN {X 0,Y 298.548,Z 119.61,A -85,B 0,C 180,E1 -16393.616,E2 -16393.616} C_VEL
LIN {X 0,Y 298.544,Z 119.606,A -85,B 0,C 180,E1 -16396.409,E2 -16396.409} C_VEL
LIN {X 0,Y 298.507,Z 119.614,A -85,B 0,C 180,E1 -16399.655,E2 -16399.655} C_VEL
LIN {X 0,Y 298.453,Z 119.618,A -85,B 0,C 180,E1 -16403.598,E2 -16403.598} C_VEL
LIN {X 0,Y 298.481,Z 119.615,A -85,B 0,C 180,E1 -16406.575,E2 -16406.575} C_VEL
LIN {X 0,Y 298.412,Z 119.623,A -85,B 0,C 180,E1 -16409.642,E2 -16409.642} C_VEL
LIN {X 0,Y 298.391,Z 119.627,A -85,B 0,C 180,E1 -16412.801,E2 -16412.801} C_VEL
LIN {X 0,Y 298.441,Z 119.623,A -85,B 0,C 180,E1 -16416.808,E2 -16416.808} C_VEL
LIN {X 0,Y 298.384,Z 119.63,A -85,B 0,C 180,E1 -16421.089,E2 -16421.089} C_VEL
LIN {X 0,Y 298.385,Z 119.628,A -85,B 0,C 180,E1 -16425.042,E2 -16425.042} C_VEL
LIN {X 0,Y 298.416,Z 119.627,A -85,B 0,C 180,E1 -16428.906,E2 -16428.906} C_VEL
LIN {X 0,Y 298.463,Z 119.616,A -85,B 0,C 180,E1 -16433.188,E2 -16433.188} C_VEL
LIN {X 0,Y 298.392,Z 119.627,A -85,B 0,C 180,E1 -16437.201,E2 -16437.201} C_VEL
LIN {X 0,Y 298.425,Z 119.624,A -85,B 0,C 180,E1 -16440.617,E2 -16440.617} C_VEL
LIN {X 0,Y 298.475,Z 119.615,A -85,B 0,C 180,E1 -16443.478,E2 -16443.478} C_VEL
LIN {X 0,Y 298.434,Z 119.623,A -85,B 0,C 180,E1 -16446.698,E2 -16446.698} C_VEL
LIN {X 0,Y 298.542,Z 119.609,A -85,B 0,C 180,E1 -16450.758,E2 -16450.758} C_VEL
LIN {X 0,Y 298.593,Z 119.599,A -85,B 0,C 180,E1 -16454.996,E2 -16454.996} C_VEL
LIN {X 0,Y 298.594,Z 119.601,A -85,B 0,C 180,E1 -16459.148,E2 -16459.148} C_VEL
LIN {X 0,Y 298.759,Z 119.581,A -85,B 0,C 180,E1 -16461.887,E2 -16461.887} C_VEL
LIN {X 0,Y 298.66,Z 119.594,A -85,B 0,C 180,E1 -16464.6,E2 -16464.6} C_VEL
LIN {X 0,Y 298.923,Z 119.561,A -85,B 0,C 180,E1 -16468.654,E2 -16468.654} C_VEL
LIN {X 0,Y 298.923,Z 119.559,A -85,B 0,C 180,E1 -16471.348,E2 -16471.348} C_VEL
LIN {X 0,Y 298.799,Z 119.576,A -85,B 0,C 180,E1 -16476.755,E2 -16476.755} C_VEL
LIN {X 0,Y 298.682,Z 119.592,A -85,B 0,C 180,E1 -16479.481,E2 -16479.481} C_VEL
LIN {X 0,Y 298.554,Z 119.608,A -85,B 0,C 180,E1 -16483.616,E2 -16483.616} C_VEL
LIN {X 0,Y 298.551,Z 119.607,A -85,B 0,C 180,E1 -16486.409,E2 -16486.409} C_VEL
LIN {X 0,Y 298.513,Z 119.614,A -85,B 0,C 180,E1 -16489.655,E2 -16489.655} C_VEL
LIN {X 0,Y 298.46,Z 119.62,A -85,B 0,C 180,E1 -16493.598,E2 -16493.598} C_VEL
LIN {X 0,Y 298.489,Z 119.614,A -85,B 0,C 180,E1 -16496.575,E2 -16496.575} C_VEL
LIN {X 0,Y 298.419,Z 119.628,A -85,B 0,C 180,E1 -16499.642,E2 -16499.642} C_VEL
LIN {X 0,Y 298.398,Z 119.626,A -85,B 0,C 180,E1 -16502.801,E2 -16502.801} C_VEL
LIN {X 0,Y 298.468,Z 119.618,A -85,B 0,C 180,E1 -16506.813,E2 -16506.813} C_VEL
LIN {X 0,Y 298.391,Z 119.628,A -85,B 0,C 180,E1 -16511.088,E2 -16511.088} C_VEL
LIN {X 0,Y 298.392,Z 119.629,A -85,B 0,C 180,E1 -16515.042,E2 -16515.042} C_VEL
LIN {X 0,Y 298.421,Z 119.626,A -85,B 0,C 180,E1 -16517.093,E2 -16517.093} C_VEL
LIN {X 0,Y 299.53,Z 122.628,A -85,B 0,C 180,E1 -16517.371,E2 -16517.371} C_VEL
LIN {X 0,Y 314.001,Z 150.358,A -85,B 0,C 180,E1 -16520.081,E2 -16520.081} C_VEL
LIN {X 0,Y 325.695,Z 174.124,A -85,B 0,C 180,E1 -16522.124,E2 -16522.124} C_VEL
LIN {X 0,Y 317.507,Z 304.949,A -85,B 0,C 180,E1 -16526.211,E2 -16526.211} C_VEL
LIN {X 0,Y 316.228,Z 322.289,A -85,B 0,C 180,E1 -16527.01,E2 -16527.01} C_VEL
LIN {X 0,Y 314.64,Z 339.781,A -85,B 0,C 180,E1 -16528.082,E2 -16528.082} C_VEL
LIN {X 0,Y 313.531,Z 349.686,A -85,B 0,C 180,E1 -16528.813,E2 -16528.813} C_VEL
LIN {X 0,Y 312.357,Z 355.044,A -85,B 0,C 180,E1 -16529.215,E2 -16529.215} C_VEL
LIN {X 0,Y 305.359,Z 370.36,A -85,B 0,C 180,E1 -16530.333,E2 -16530.333} C_VEL
LIN {X 0,Y 303.65,Z 375.431,A -85,B 0,C 180,E1 -16530.818,E2 -16530.818} C_VEL
LIN {X 0,Y 303.331,Z 377.095,A -85,B 0,C 180,E1 -16531.004,E2 -16531.004} C_VEL
LIN {X 0,Y 301.305,Z 390.836,A -85,B 0,C 180,E1 -16532.677,E2 -16532.677} C_VEL
LIN {X 0,Y 299.033,Z 405.367,A -85,B 0,C 180,E1 -16534.787,E2 -16534.787} C_VEL
LIN {X 0,Y 296.875,Z 418.634,A -85,B 0,C 180,E1 -16537.081,E2 -16537.081} C_VEL
LIN {X 0,Y 295.198,Z 430.097,A -85,B 0,C 180,E1 -16539.441,E2 -16539.441} C_VEL
LIN {X 0,Y 293.382,Z 441.495,A -85,B 0,C 180,E1 -16542.216,E2 -16542.216} C_VEL
LIN {X 0,Y 292.314,Z 449.888,A -85,B 0,C 180,E1 -16544.664,E2 -16544.664} C_VEL
LIN {X 0,Y 291.196,Z 457.969,A -85,B 0,C 180,E1 -16547.454,E2 -16547.454} C_VEL
LIN {X 0,Y 290.617,Z 464.642,A -85,B 0,C 180,E1 -16550.254,E2 -16550.254} C_VEL
LIN {X 0,Y 290.24,Z 470.076,A -85,B 0,C 180,E1 -16553.122,E2 -16553.122} C_VEL
LIN {X 0,Y 290.01,Z 474.049,A -85,B 0,C 180,E1 -16555.831,E2 -16555.831} C_VEL
LIN {X 0,Y 290.008,Z 477.099,A -85,B 0,C 180,E1 -16558.611,E2 -16558.611} C_VEL
LIN {X 0,Y 290.173,Z 479.001,A -85,B 0,C 180,E1 -16561.388,E2 -16561.388} C_VEL
LIN {X 0,Y 290.597,Z 479.938,A -85,B 0,C 180,E1 -16564.161,E2 -16564.161} C_VEL
LIN {X 0,Y 290.986,Z 479.862,A -85,B 0,C 180,E1 -16566.936,E2 -16566.936} C_VEL
LIN {X 0,Y 292.063,Z 478.767,A -85,B 0,C 180,E1 -16569.697,E2 -16569.697} C_VEL
LIN {X 0,Y 293.312,Z 476.721,A -85,B 0,C 180,E1 -16572.453,E2 -16572.453} C_VEL
LIN {X 0,Y 295.04,Z 473.635,A -85,B 0,C 180,E1 -16575.19,E2 -16575.19} C_VEL
LIN {X 0,Y 297.192,Z 469.605,A -85,B 0,C 180,E1 -16577.904,E2 -16577.904} C_VEL
LIN {X 0,Y 300.01,Z 464.386,A -85,B 0,C 180,E1 -16580.572,E2 -16580.572} C_VEL
LIN {X 0,Y 303.309,Z 458.101,A -85,B 0,C 180,E1 -16583.198,E2 -16583.198} C_VEL
LIN {X 0,Y 307.778,Z 449.538,A -85,B 0,C 180,E1 -16586.076,E2 -16586.076} C_VEL
LIN {X 0,Y 312.811,Z 439.547,A -85,B 0,C 180,E1 -16588.809,E2 -16588.809} C_VEL
LIN {X 0,Y 318.168,Z 428.599,A -85,B 0,C 180,E1 -16591.271,E2 -16591.271} C_VEL
LIN {X 0,Y 324.102,Z 416.098,A -85,B 0,C 180,E1 -16593.57,E2 -16593.57} C_VEL
LIN {X 0,Y 329.535,Z 403.961,A -85,B 0,C 180,E1 -16595.466,E2 -16595.466} C_VEL
LIN {X 0,Y 335.856,Z 389.171,A -85,B 0,C 180,E1 -16597.361,E2 -16597.361} C_VEL
LIN {X 0,Y 342.58,Z 372.262,A -85,B 0,C 180,E1 -16599.111,E2 -16599.111} C_VEL
LIN {X 0,Y 348.744,Z 355.228,A -85,B 0,C 180,E1 -16600.535,E2 -16600.535} C_VEL
LIN {X 0,Y 354.209,Z 338.237,A -85,B 0,C 180,E1 -16601.658,E2 -16601.658} C_VEL
LIN {X 0,Y 358.836,Z 321.518,A -85,B 0,C 180,E1 -16602.508,E2 -16602.508} C_VEL
LIN {X 0,Y 367.265,Z 288.386,A -85,B 0,C 180,E1 -16603.779,E2 -16603.779} C_VEL
LIN {X 0,Y 371.845,Z 271.281,A -85,B 0,C 180,E1 -16604.402,E2 -16604.402} C_VEL
LIN {X 0,Y 369.719,Z 279.413,A -85,B 0,C 180,E1 -16604.726,E2 -16604.726} C_VEL
LIN {X 0,Y 355.017,Z 337.955,A -85,B 0,C 180,E1 -16606.923,E2 -16606.923} C_VEL
LIN {X 0,Y 349.871,Z 355.201,A -85,B 0,C 180,E1 -16607.706,E2 -16607.706} C_VEL
LIN {X 0,Y 343.67,Z 373.477,A -85,B 0,C 180,E1 -16608.737,E2 -16608.737} C_VEL
LIN {X 0,Y 337.77,Z 389.296,A -85,B 0,C 180,E1 -16609.832,E2 -16609.832} C_VEL
LIN {X 0,Y 331.88,Z 404.374,A -85,B 0,C 180,E1 -16611.144,E2 -16611.144} C_VEL
LIN {X 0,Y 325.027,Z 421.157,A -85,B 0,C 180,E1 -16612.933,E2 -16612.933} C_VEL
LIN {X 0,Y 318.444,Z 436.837,A -85,B 0,C 180,E1 -16614.982,E2 -16614.982} C_VEL
LIN {X 0,Y 312.961,Z 449.693,A -85,B 0,C 180,E1 -16617.004,E2 -16617.004} C_VEL
LIN {X 0,Y 307.522,Z 462.679,A -85,B 0,C 180,E1 -16619.436,E2 -16619.436} C_VEL
LIN {X 0,Y 302.337,Z 475.377,A -85,B 0,C 180,E1 -16622.295,E2 -16622.295} C_VEL
LIN {X 0,Y 298.231,Z 486.247,A -85,B 0,C 180,E1 -16625.272,E2 -16625.272} C_VEL
LIN {X 0,Y 294.963,Z 495.475,A -85,B 0,C 180,E1 -16628.316,E2 -16628.316} C_VEL
LIN {X 0,Y 292.725,Z 502.432,A -85,B 0,C 180,E1 -16631.087,E2 -16631.087} C_VEL
LIN {X 0,Y 291.206,Z 508.203,A -85,B 0,C 180,E1 -16633.885,E2 -16633.885} C_VEL
LIN {X 0,Y 290.228,Z 512.934,A -85,B 0,C 180,E1 -16636.699,E2 -16636.699} C_VEL
LIN {X 0,Y 289.734,Z 515.76,A -85,B 0,C 180,E1 -16638.81,E2 -16638.81} C_VEL
LIN {X 0,Y 289.654,Z 518.549,A -85,B 0,C 180,E1 -16641.628,E2 -16641.628} C_VEL
LIN {X 0,Y 289.779,Z 520.356,A -85,B 0,C 180,E1 -16644.432,E2 -16644.432} C_VEL
LIN {X 0,Y 289.934,Z 520.98,A -85,B 0,C 180,E1 -16647.22,E2 -16647.22} C_VEL
LIN {X 0,Y 290.196,Z 520.543,A -85,B 0,C 180,E1 -16649.999,E2 -16649.999} C_VEL
LIN {X 0,Y 290.108,Z 518.86,A -85,B 0,C 180,E1 -16652.776,E2 -16652.776} C_VEL
LIN {X 0,Y 290.001,Z 515.968,A -85,B 0,C 180,E1 -16655.562,E2 -16655.562} C_VEL
LIN {X 0,Y 289.995,Z 512.969,A -85,B 0,C 180,E1 -16657.659,E2 -16657.659} C_VEL
LIN {X 0,Y 289.964,Z 507.78,A -85,B 0,C 180,E1 -16660.473,E2 -16660.473} C_VEL
LIN {X 0,Y 290.348,Z 501.224,A -85,B 0,C 180,E1 -16663.293,E2 -16663.293} C_VEL
LIN {X 0,Y 291.025,Z 493.055,A -85,B 0,C 180,E1 -16666.123,E2 -16666.123} C_VEL
LIN {X 0,Y 292.171,Z 483.138,A -85,B 0,C 180,E1 -16668.948,E2 -16668.948} C_VEL
LIN {X 0,Y 293.569,Z 472.791,A -85,B 0,C 180,E1 -16671.412,E2 -16671.412} C_VEL
LIN {X 0,Y 295.165,Z 462.532,A -85,B 0,C 180,E1 -16673.504,E2 -16673.504} C_VEL
LIN {X 0,Y 297.256,Z 449.552,A -85,B 0,C 180,E1 -16675.758,E2 -16675.758} C_VEL
LIN {X 0,Y 299.52,Z 435.585,A -85,B 0,C 180,E1 -16677.797,E2 -16677.797} C_VEL
LIN {X 0,Y 301.93,Z 420.355,A -85,B 0,C 180,E1 -16679.645,E2 -16679.645} C_VEL
LIN {X 0,Y 304.493,Z 403.646,A -85,B 0,C 180,E1 -16681.3,E2 -16681.3} C_VEL
LIN {X 0,Y 306.756,Z 386.472,A -85,B 0,C 180,E1 -16682.671,E2 -16682.671} C_VEL
LIN {X 0,Y 308.711,Z 369.985,A -85,B 0,C 180,E1 -16683.704,E2 -16683.704} C_VEL
LIN {X 0,Y 310.546,Z 351.796,A -85,B 0,C 180,E1 -16684.553,E2 -16684.553} C_VEL
LIN {X 0,Y 320.502,Z 201.606,A -85,B 0,C 180,E1 -16689.408,E2 -16689.408} C_VEL
LIN {X 0,Y 318.852,Z 186.929,A -85,B 0,C 180,E1 -16690.132,E2 -16690.132} C_VEL
LIN {X 0,Y 304.424,Z 154.423,A -85,B 0,C 180,E1 -16692.94,E2 -16692.94} C_VEL
LIN {X 0,Y 298.404,Z 141.463,A -85,B 0,C 180,E1 -16694.204,E2 -16694.204} C_VEL
LIN {X 0,Y 292.067,Z 122.759,A -85,B 0,C 180,E1 -16698.141,E2 -16698.141} C_VEL
LIN {X 0,Y 291.364,Z 120.506,A -85,B 0,C 180,E1 -16698.662,E2 -16698.662} C_VEL
LIN {X 0,Y 291.421,Z 120.496,A -85,B 0,C 180,E1 -16702.922,E2 -16702.922} C_VEL
LIN {X 0,Y 291.341,Z 120.508,A -85,B 0,C 180,E1 -16706.301,E2 -16706.301} C_VEL
LIN {X 0,Y 291.383,Z 120.504,A -85,B 0,C 180,E1 -16710.259,E2 -16710.259} C_VEL
LIN {X 0,Y 291.413,Z 120.501,A -85,B 0,C 180,E1 -16714.272,E2 -16714.272} C_VEL
LIN {X 0,Y 291.377,Z 120.502,A -85,B 0,C 180,E1 -16717.299,E2 -16717.299} C_VEL
LIN {X 0,Y 291.453,Z 120.494,A -85,B 0,C 180,E1 -16720.27,E2 -16720.27} C_VEL
LIN {X 0,Y 291.55,Z 120.479,A -85,B 0,C 180,E1 -16724.624,E2 -16724.624} C_VEL
LIN {X 0,Y 291.534,Z 120.478,A -85,B 0,C 180,E1 -16728.881,E2 -16728.881} C_VEL
LIN {X 0,Y 291.705,Z 120.464,A -85,B 0,C 180,E1 -16731.689,E2 -16731.689} C_VEL
LIN {X 0,Y 291.627,Z 120.465,A -85,B 0,C 180,E1 -16734.468,E2 -16734.468} C_VEL
LIN {X 0,Y 291.886,Z 120.437,A -85,B 0,C 180,E1 -16738.62,E2 -16738.62} C_VEL
LIN {X 0,Y 291.886,Z 120.439,A -85,B 0,C 180,E1 -16741.38,E2 -16741.38} C_VEL
LIN {X 0,Y 291.743,Z 120.454,A -85,B 0,C 180,E1 -16746.918,E2 -16746.918} C_VEL
LIN {X 0,Y 291.625,Z 120.471,A -85,B 0,C 180,E1 -16749.712,E2 -16749.712} C_VEL
LIN {X 0,Y 291.518,Z 120.483,A -85,B 0,C 180,E1 -16753.951,E2 -16753.951} C_VEL
LIN {X 0,Y 291.483,Z 120.487,A -85,B 0,C 180,E1 -16756.818,E2 -16756.818} C_VEL
LIN {X 0,Y 291.446,Z 120.492,A -85,B 0,C 180,E1 -16759.875,E2 -16759.875} C_VEL
LIN {X 0,Y 291.395,Z 120.495,A -85,B 0,C 180,E1 -16764.206,E2 -16764.206} C_VEL
LIN {X 0,Y 291.415,Z 120.499,A -85,B 0,C 180,E1 -16767.272,E2 -16767.272} C_VEL
LIN {X 0,Y 291.33,Z 120.504,A -85,B 0,C 180,E1 -16770.438,E2 -16770.438} C_VEL
LIN {X 0,Y 291.341,Z 120.505,A -85,B 0,C 180,E1 -16773.699,E2 -16773.699} C_VEL
LIN {X 0,Y 291.369,Z 120.501,A -85,B 0,C 180,E1 -16777.254,E2 -16777.254} C_VEL
LIN {X 0,Y 291.329,Z 120.507,A -85,B 0,C 180,E1 -16780.643,E2 -16780.643} C_VEL
LIN {X 0,Y 291.311,Z 120.509,A -85,B 0,C 180,E1 -16784.398,E2 -16784.398} C_VEL
LIN {X 0,Y 291.353,Z 120.503,A -85,B 0,C 180,E1 -16788.398,E2 -16788.398} C_VEL
LIN {X 0,Y 291.372,Z 120.501,A -85,B 0,C 180,E1 -16791.163,E2 -16791.163} C_VEL
LIN {X 0,Y 291.383,Z 120.5,A -85,B 0,C 180,E1 -16794.63,E2 -16794.63} C_VEL
LIN {X 0,Y 291.368,Z 120.501,A -85,B 0,C 180,E1 -16797.951,E2 -16797.951} C_VEL
LIN {X 0,Y 291.374,Z 120.498,A -85,B 0,C 180,E1 -16801.159,E2 -16801.159} C_VEL
LIN {X 0,Y 291.411,Z 120.498,A -85,B 0,C 180,E1 -16804.273,E2 -16804.273} C_VEL
LIN {X 0,Y 291.389,Z 120.497,A -85,B 0,C 180,E1 -16807.301,E2 -16807.301} C_VEL
LIN {X 0,Y 291.462,Z 120.491,A -85,B 0,C 180,E1 -16810.272,E2 -16810.272} C_VEL
LIN {X 0,Y 291.555,Z 120.478,A -85,B 0,C 180,E1 -16814.625,E2 -16814.625} C_VEL
LIN {X 0,Y 291.537,Z 120.48,A -85,B 0,C 180,E1 -16818.882,E2 -16818.882} C_VEL
LIN {X 0,Y 291.709,Z 120.458,A -85,B 0,C 180,E1 -16821.689,E2 -16821.689} C_VEL
LIN {X 0,Y 291.631,Z 120.47,A -85,B 0,C 180,E1 -16824.469,E2 -16824.469} C_VEL
LIN {X 0,Y 291.889,Z 120.437,A -85,B 0,C 180,E1 -16828.621,E2 -16828.621} C_VEL
LIN {X 0,Y 291.889,Z 120.436,A -85,B 0,C 180,E1 -16831.381,E2 -16831.381} C_VEL
LIN {X 0,Y 291.748,Z 120.454,A -85,B 0,C 180,E1 -16836.919,E2 -16836.919} C_VEL
LIN {X 0,Y 291.631,Z 120.472,A -85,B 0,C 180,E1 -16839.713,E2 -16839.713} C_VEL
LIN {X 0,Y 291.524,Z 120.487,A -85,B 0,C 180,E1 -16843.951,E2 -16843.951} C_VEL
LIN {X 0,Y 291.489,Z 120.486,A -85,B 0,C 180,E1 -16846.819,E2 -16846.819} C_VEL
LIN {X 0,Y 291.453,Z 120.494,A -85,B 0,C 180,E1 -16849.876,E2 -16849.876} C_VEL
LIN {X 0,Y 291.403,Z 120.498,A -85,B 0,C 180,E1 -16854.206,E2 -16854.206} C_VEL
LIN {X 0,Y 291.422,Z 120.497,A -85,B 0,C 180,E1 -16857.272,E2 -16857.272} C_VEL
LIN {X 0,Y 291.337,Z 120.506,A -85,B 0,C 180,E1 -16860.438,E2 -16860.438} C_VEL
LIN {X 0,Y 291.347,Z 120.507,A -85,B 0,C 180,E1 -16863.699,E2 -16863.699} C_VEL
LIN {X 0,Y 291.397,Z 120.501,A -85,B 0,C 180,E1 -16867.259,E2 -16867.259} C_VEL
LIN {X 0,Y 291.338,Z 120.505,A -85,B 0,C 180,E1 -16870.643,E2 -16870.643} C_VEL
LIN {X 0,Y 291.317,Z 120.509,A -85,B 0,C 180,E1 -16874.398,E2 -16874.398} C_VEL
LIN {X 0,Y 291.341,Z 120.522,A -85,B 0,C 180,E1 -16876.306,E2 -16876.306} C_VEL
LIN {X 0,Y 292.353,Z 123.362,A -85,B 0,C 180,E1 -16876.553,E2 -16876.553} C_VEL
LIN {X 0,Y 300.287,Z 138.27,A -85,B 0,C 180,E1 -16878.122,E2 -16878.122} C_VEL
LIN {X 0,Y 313.52,Z 164.366,A -85,B 0,C 180,E1 -16880.581,E2 -16880.581} C_VEL
LIN {X 0,Y 319.287,Z 176.277,A -85,B 0,C 180,E1 -16881.603,E2 -16881.603} C_VEL
LIN {X 0,Y 310.909,Z 305.173,A -85,B 0,C 180,E1 -16885.737,E2 -16885.737} C_VEL
LIN {X 0,Y 309.531,Z 323.221,A -85,B 0,C 180,E1 -16886.592,E2 -16886.592} C_VEL
LIN {X 0,Y 307.82,Z 341.41,A -85,B 0,C 180,E1 -16887.747,E2 -16887.747} C_VEL
LIN {X 0,Y 305.938,Z 357.871,A -85,B 0,C 180,E1 -16889.069,E2 -16889.069} C_VEL
LIN {X 0,Y 303.663,Z 374.706,A -85,B 0,C 180,E1 -16890.73,E2 -16890.73} C_VEL
LIN {X 0,Y 303.331,Z 377.095,A -85,B 0,C 180,E1 -16891.004,E2 -16891.004} C_VEL
LIN {X 0,Y 302.005,Z 382.139,A -85,B 0,C 180,E1 -16891.546,E2 -16891.546} C_VEL
LIN {X 0,Y 298.089,Z 390.135,A -85,B 0,C 180,E1 -16892.397,E2 -16892.397} C_VEL
LIN {X 0,Y 294.089,Z 397.847,A -85,B 0,C 180,E1 -16893.32,E2 -16893.32} C_VEL
LIN {X 0,Y 292.624,Z 402.388,A -85,B 0,C 180,E1 -16893.978,E2 -16893.978} C_VEL
LIN {X 0,Y 290.573,Z 414.985,A -85,B 0,C 180,E1 -16896.101,E2 -16896.101} C_VEL
LIN {X 0,Y 288.636,Z 427.419,A -85,B 0,C 180,E1 -16898.578,E2 -16898.578} C_VEL
LIN {X 0,Y 286.933,Z 438.015,A -85,B 0,C 180,E1 -16901.062,E2 -16901.062} C_VEL
LIN {X 0,Y 285.599,Z 447.441,A -85,B 0,C 180,E1 -16903.683,E2 -16903.683} C_VEL
LIN {X 0,Y 284.461,Z 455.708,A -85,B 0,C 180,E1 -16906.425,E2 -16906.425} C_VEL
LIN {X 0,Y 283.68,Z 462.867,A -85,B 0,C 180,E1 -16909.292,E2 -16909.292} C_VEL
LIN {X 0,Y 283.242,Z 468.712,A -85,B 0,C 180,E1 -16912.156,E2 -16912.156} C_VEL
LIN {X 0,Y 282.954,Z 473.28,A -85,B 0,C 180,E1 -16915.013,E2 -16915.013} C_VEL
LIN {X 0,Y 282.916,Z 475.98,A -85,B 0,C 180,E1 -16917.152,E2 -16917.152} C_VEL
LIN {X 0,Y 282.981,Z 478.554,A -85,B 0,C 180,E1 -16920,E2 -16920} C_VEL
LIN {X 0,Y 283.319,Z 480.148,A -85,B 0,C 180,E1 -16922.844,E2 -16922.844} C_VEL
LIN {X 0,Y 283.755,Z 480.71,A -85,B 0,C 180,E1 -16925.686,E2 -16925.686} C_VEL
LIN {X 0,Y 284.741,Z 480.057,A -85,B 0,C 180,E1 -16929.143,E2 -16929.143} C_VEL
LIN {X 0,Y 285.738,Z 478.894,A -85,B 0,C 180,E1 -16931.348,E2 -16931.348} C_VEL
LIN {X 0,Y 287.31,Z 476.493,A -85,B 0,C 180,E1 -16934.159,E2 -16934.159} C_VEL
LIN {X 0,Y 289.337,Z 473.171,A -85,B 0,C 180,E1 -16936.946,E2 -16936.946} C_VEL
LIN {X 0,Y 292.587,Z 467.791,A -85,B 0,C 180,E1 -16940.204,E2 -16940.204} C_VEL
LIN {X 0,Y 297.08,Z 460.133,A -85,B 0,C 180,E1 -16943.714,E2 -16943.714} C_VEL
LIN {X 0,Y 302.368,Z 450.888,A -85,B 0,C 180,E1 -16946.952,E2 -16946.952} C_VEL
LIN {X 0,Y 307.992,Z 440.645,A -85,B 0,C 180,E1 -16949.829,E2 -16949.829} C_VEL
LIN {X 0,Y 313.439,Z 430.484,A -85,B 0,C 180,E1 -16952.176,E2 -16952.176} C_VEL
LIN {X 0,Y 319.711,Z 418.389,A -85,B 0,C 180,E1 -16954.475,E2 -16954.475} C_VEL
LIN {X 0,Y 325.948,Z 405.647,A -85,B 0,C 180,E1 -16956.514,E2 -16956.514} C_VEL
LIN {X 0,Y 333.075,Z 390.358,A -85,B 0,C 180,E1 -16958.496,E2 -16958.496} C_VEL
LIN {X 0,Y 340.202,Z 373.925,A -85,B 0,C 180,E1 -16960.208,E2 -16960.208} C_VEL
LIN {X 0,Y 347.297,Z 355.911,A -85,B 0,C 180,E1 -16961.702,E2 -16961.702} C_VEL
LIN {X 0,Y 353.075,Z 339.293,A -85,B 0,C 180,E1 -16962.786,E2 -16962.786} C_VEL
LIN {X 0,Y 357.755,Z 323.671,A -85,B 0,C 180,E1 -16963.583,E2 -16963.583} C_VEL
LIN {X 0,Y 363.411,Z 302.648,A -85,B 0,C 180,E1 -16964.401,E2 -16964.401} C_VEL
LIN {X 0,Y 363.25,Z 303.257,A -85,B 0,C 180,E1 -16964.463,E2 -16964.463} C_VEL
LIN {X 0,Y 354.251,Z 336.855,A -85,B 0,C 180,E1 -16965.725,E2 -16965.725} C_VEL
LIN {X 0,Y 348.219,Z 355.568,A -85,B 0,C 180,E1 -16966.561,E2 -16966.561} C_VEL
LIN {X 0,Y 342.016,Z 372.466,A -85,B 0,C 180,E1 -16967.503,E2 -16967.503} C_VEL
LIN {X 0,Y 335.197,Z 389.375,A -85,B 0,C 180,E1 -16968.665,E2 -16968.665} C_VEL
LIN {X 0,Y 329.007,Z 403.983,A -85,B 0,C 180,E1 -16969.945,E2 -16969.945} C_VEL
LIN {X 0,Y 321.719,Z 420.371,A -85,B 0,C 180,E1 -16971.693,E2 -16971.693} C_VEL
LIN {X 0,Y 314.693,Z 435.802,A -85,B 0,C 180,E1 -16973.727,E2 -16973.727} C_VEL
LIN {X 0,Y 308.03,Z 450.148,A -85,B 0,C 180,E1 -16976.013,E2 -16976.013} C_VEL
LIN {X 0,Y 301.591,Z 464.274,A -85,B 0,C 180,E1 -16978.768,E2 -16978.768} C_VEL
LIN {X 0,Y 296.143,Z 476.479,A -85,B 0,C 180,E1 -16981.663,E2 -16981.663} C_VEL
LIN {X 0,Y 291.806,Z 486.945,A -85,B 0,C 180,E1 -16984.69,E2 -16984.69} C_VEL
LIN {X 0,Y 288.192,Z 496.186,A -85,B 0,C 180,E1 -16987.924,E2 -16987.924} C_VEL
LIN {X 0,Y 285.453,Z 504.071,A -85,B 0,C 180,E1 -16991.332,E2 -16991.332} C_VEL
LIN {X 0,Y 284.011,Z 509.455,A -85,B 0,C 180,E1 -16994.204,E2 -16994.204} C_VEL
LIN {X 0,Y 283.011,Z 513.674,A -85,B 0,C 180,E1 -16997.085,E2 -16997.085} C_VEL
LIN {X 0,Y 282.557,Z 516.943,A -85,B 0,C 180,E1 -16999.972,E2 -16999.972} C_VEL
LIN {X 0,Y 282.602,Z 519.073,A -85,B 0,C 180,E1 -17002.856,E2 -17002.856} C_VEL
LIN {X 0,Y 282.697,Z 519.778,A -85,B 0,C 180,E1 -17004.292,E2 -17004.292} C_VEL
LIN {X 0,Y 282.848,Z 520.333,A -85,B 0,C 180,E1 -17007.151,E2 -17007.151} C_VEL
LIN {X 0,Y 283.163,Z 519.746,A -85,B 0,C 180,E1 -17009.999,E2 -17009.999} C_VEL
LIN {X 0,Y 283.053,Z 517.996,A -85,B 0,C 180,E1 -17012.845,E2 -17012.845} C_VEL
LIN {X 0,Y 282.957,Z 514.941,A -85,B 0,C 180,E1 -17015.701,E2 -17015.701} C_VEL
LIN {X 0,Y 282.926,Z 511.853,A -85,B 0,C 180,E1 -17017.851,E2 -17017.851} C_VEL
LIN {X 0,Y 282.927,Z 506.488,A -85,B 0,C 180,E1 -17020.736,E2 -17020.736} C_VEL
LIN {X 0,Y 283.34,Z 499.737,A -85,B 0,C 180,E1 -17023.628,E2 -17023.628} C_VEL
LIN {X 0,Y 284.09,Z 491.407,A -85,B 0,C 180,E1 -17026.528,E2 -17026.528} C_VEL
LIN {X 0,Y 285.125,Z 482.629,A -85,B 0,C 180,E1 -17029.061,E2 -17029.061} C_VEL
LIN {X 0,Y 286.556,Z 472.278,A -85,B 0,C 180,E1 -17031.584,E2 -17031.584} C_VEL
LIN {X 0,Y 288.189,Z 462.016,A -85,B 0,C 180,E1 -17033.726,E2 -17033.726} C_VEL
LIN {X 0,Y 290.347,Z 448.874,A -85,B 0,C 180,E1 -17036.058,E2 -17036.058} C_VEL
LIN {X 0,Y 292.628,Z 435.049,A -85,B 0,C 180,E1 -17038.12,E2 -17038.12} C_VEL
LIN {X 0,Y 295.117,Z 419.849,A -85,B 0,C 180,E1 -17040.005,E2 -17040.005} C_VEL
LIN {X 0,Y 297.644,Z 403.759,A -85,B 0,C 180,E1 -17041.644,E2 -17041.644} C_VEL
LIN {X 0,Y 299.872,Z 387.176,A -85,B 0,C 180,E1 -17043.017,E2 -17043.017} C_VEL
LIN {X 0,Y 302.038,Z 369.692,A -85,B 0,C 180,E1 -17044.148,E2 -17044.148} C_VEL
LIN {X 0,Y 303.894,Z 351.718,A -85,B 0,C 180,E1 -17045.016,E2 -17045.016} C_VEL
LIN {X 0,Y 313.424,Z 212.619,A -85,B 0,C 180,E1 -17049.652,E2 -17049.652} C_VEL
LIN {X 0,Y 314.111,Z 201.918,A -85,B 0,C 180,E1 -17050.007,E2 -17050.007} C_VEL
LIN {X 0,Y 312.703,Z 189.456,A -85,B 0,C 180,E1 -17050.634,E2 -17050.634} C_VEL
LIN {X 0,Y 298.623,Z 157.587,A -85,B 0,C 180,E1 -17053.457,E2 -17053.457} C_VEL
LIN {X 0,Y 290.999,Z 141.024,A -85,B 0,C 180,E1 -17055.103,E2 -17055.103} C_VEL
LIN {X 0,Y 285.191,Z 124.171,A -85,B 0,C 180,E1 -17058.761,E2 -17058.761} C_VEL
LIN {X 0,Y 284.309,Z 121.384,A -85,B 0,C 180,E1 -17059.426,E2 -17059.426} C_VEL
LIN {X 0,Y 284.346,Z 121.377,A -85,B 0,C 180,E1 -17063.616,E2 -17063.616} C_VEL
LIN {X 0,Y 284.304,Z 121.382,A -85,B 0,C 180,E1 -17067.189,E2 -17067.189} C_VEL
LIN {X 0,Y 284.355,Z 121.378,A -85,B 0,C 180,E1 -17070.376,E2 -17070.376} C_VEL
LIN {X 0,Y 284.374,Z 121.375,A -85,B 0,C 180,E1 -17073.586,E2 -17073.586} C_VEL
LIN {X 0,Y 284.362,Z 121.376,A -85,B 0,C 180,E1 -17076.707,E2 -17076.707} C_VEL
LIN {X 0,Y 284.399,Z 121.371,A -85,B 0,C 180,E1 -17081.262,E2 -17081.262} C_VEL
LIN {X 0,Y 284.488,Z 121.359,A -85,B 0,C 180,E1 -17084.459,E2 -17084.459} C_VEL
LIN {X 0,Y 284.486,Z 121.356,A -85,B 0,C 180,E1 -17088.602,E2 -17088.602} C_VEL
LIN {X 0,Y 284.655,Z 121.34,A -85,B 0,C 180,E1 -17091.481,E2 -17091.481} C_VEL
LIN {X 0,Y 284.597,Z 121.34,A -85,B 0,C 180,E1 -17094.331,E2 -17094.331} C_VEL
LIN {X 0,Y 284.852,Z 121.313,A -85,B 0,C 180,E1 -17098.586,E2 -17098.586} C_VEL
LIN {X 0,Y 284.852,Z 121.316,A -85,B 0,C 180,E1 -17101.414,E2 -17101.414} C_VEL
LIN {X 0,Y 284.695,Z 121.332,A -85,B 0,C 180,E1 -17107.09,E2 -17107.09} C_VEL
LIN {X 0,Y 284.562,Z 121.349,A -85,B 0,C 180,E1 -17109.956,E2 -17109.956} C_VEL
LIN {X 0,Y 284.478,Z 121.359,A -85,B 0,C 180,E1 -17114.303,E2 -17114.303} C_VEL
LIN {X 0,Y 284.421,Z 121.368,A -85,B 0,C 180,E1 -17117.249,E2 -17117.249} C_VEL
LIN {X 0,Y 284.375,Z 121.372,A -85,B 0,C 180,E1 -17120.243,E2 -17120.243} C_VEL
LIN {X 0,Y 284.365,Z 121.371,A -85,B 0,C 180,E1 -17123.876,E2 -17123.876} C_VEL
LIN {X 0,Y 284.39,Z 121.375,A -85,B 0,C 180,E1 -17127.173,E2 -17127.173} C_VEL
LIN {X 0,Y 284.29,Z 121.384,A -85,B 0,C 180,E1 -17131.275,E2 -17131.275} C_VEL
LIN {X 0,Y 284.337,Z 121.379,A -85,B 0,C 180,E1 -17135.349,E2 -17135.349} C_VEL
LIN {X 0,Y 284.305,Z 121.378,A -85,B 0,C 180,E1 -17138.17,E2 -17138.17} C_VEL
LIN {X 0,Y 284.266,Z 121.386,A -85,B 0,C 180,E1 -17142.125,E2 -17142.125} C_VEL
LIN {X 0,Y 284.285,Z 121.381,A -85,B 0,C 180,E1 -17146.197,E2 -17146.197} C_VEL
LIN {X 0,Y 284.349,Z 121.375,A -85,B 0,C 180,E1 -17150.014,E2 -17150.014} C_VEL
LIN {X 0,Y 284.349,Z 121.372,A -85,B 0,C 180,E1 -17153.618,E2 -17153.618} C_VEL
LIN {X 0,Y 284.305,Z 121.382,A -85,B 0,C 180,E1 -17157.191,E2 -17157.191} C_VEL
LIN {X 0,Y 284.353,Z 121.377,A -85,B 0,C 180,E1 -17160.377,E2 -17160.377} C_VEL
LIN {X 0,Y 284.373,Z 121.371,A -85,B 0,C 180,E1 -17163.587,E2 -17163.587} C_VEL
LIN {X 0,Y 284.368,Z 121.375,A -85,B 0,C 180,E1 -17166.708,E2 -17166.708} C_VEL
LIN {X 0,Y 284.405,Z 121.368,A -85,B 0,C 180,E1 -17171.263,E2 -17171.263} C_VEL
LIN {X 0,Y 284.492,Z 121.359,A -85,B 0,C 180,E1 -17174.46,E2 -17174.46} C_VEL
LIN {X 0,Y 284.489,Z 121.36,A -85,B 0,C 180,E1 -17178.602,E2 -17178.602} C_VEL
LIN {X 0,Y 284.659,Z 121.335,A -85,B 0,C 180,E1 -17181.482,E2 -17181.482} C_VEL
LIN {X 0,Y 284.602,Z 121.347,A -85,B 0,C 180,E1 -17184.332,E2 -17184.332} C_VEL
LIN {X 0,Y 284.855,Z 121.314,A -85,B 0,C 180,E1 -17188.587,E2 -17188.587} C_VEL
LIN {X 0,Y 284.855,Z 121.312,A -85,B 0,C 180,E1 -17191.415,E2 -17191.415} C_VEL
LIN {X 0,Y 284.7,Z 121.332,A -85,B 0,C 180,E1 -17197.091,E2 -17197.091} C_VEL
LIN {X 0,Y 284.568,Z 121.35,A -85,B 0,C 180,E1 -17199.956,E2 -17199.956} C_VEL
LIN {X 0,Y 284.484,Z 121.361,A -85,B 0,C 180,E1 -17204.304,E2 -17204.304} C_VEL
LIN {X 0,Y 284.427,Z 121.367,A -85,B 0,C 180,E1 -17207.249,E2 -17207.249} C_VEL
LIN {X 0,Y 284.382,Z 121.373,A -85,B 0,C 180,E1 -17210.243,E2 -17210.243} C_VEL
LIN {X 0,Y 284.372,Z 121.375,A -85,B 0,C 180,E1 -17213.876,E2 -17213.876} C_VEL
LIN {X 0,Y 284.398,Z 121.371,A -85,B 0,C 180,E1 -17217.174,E2 -17217.174} C_VEL
LIN {X 0,Y 284.296,Z 121.385,A -85,B 0,C 180,E1 -17221.275,E2 -17221.275} C_VEL
LIN {X 0,Y 284.365,Z 121.376,A -85,B 0,C 180,E1 -17225.355,E2 -17225.355} C_VEL
LIN {X 0,Y 284.326,Z 121.379,A -85,B 0,C 180,E1 -17228.168,E2 -17228.168} C_VEL
LIN {X 0,Y 284.273,Z 121.386,A -85,B 0,C 180,E1 -17232.125,E2 -17232.125} C_VEL
LIN {X 0,Y 284.271,Z 121.419,A -85,B 0,C 180,E1 -17235.478,E2 -17235.478} C_VEL
LIN {X 0,Y 285.279,Z 124.231,A -85,B 0,C 180,E1 -17235.735,E2 -17235.735} C_VEL
LIN {X 0,Y 296.252,Z 144.831,A -85,B 0,C 180,E1 -17237.95,E2 -17237.95} C_VEL
LIN {X 0,Y 310.549,Z 173.503,A -85,B 0,C 180,E1 -17240.647,E2 -17240.647} C_VEL
LIN {X 0,Y 312.803,Z 178.165,A -85,B 0,C 180,E1 -17241.052,E2 -17241.052} C_VEL
LIN {X 0,Y 304.252,Z 305.987,A -85,B 0,C 180,E1 -17245.282,E2 -17245.282} C_VEL
LIN {X 0,Y 302.858,Z 323.907,A -85,B 0,C 180,E1 -17246.156,E2 -17246.156} C_VEL
LIN {X 0,Y 301.217,Z 340.838,A -85,B 0,C 180,E1 -17247.249,E2 -17247.249} C_VEL
LIN {X 0,Y 299.385,Z 356.487,A -85,B 0,C 180,E1 -17248.512,E2 -17248.512} C_VEL
LIN {X 0,Y 297.264,Z 372.055,A -85,B 0,C 180,E1 -17250.037,E2 -17250.037} C_VEL
LIN {X 0,Y 294.956,Z 387.332,A -85,B 0,C 180,E1 -17251.839,E2 -17251.839} C_VEL
LIN {X 0,Y 292.805,Z 401.419,A -85,B 0,C 180,E1 -17253.83,E2 -17253.83} C_VEL
LIN {X 0,Y 292.624,Z 402.388,A -85,B 0,C 180,E1 -17253.978,E2 -17253.978} C_VEL
LIN {X 0,Y 291.185,Z 406.951,A -85,B 0,C 180,E1 -17254.665,E2 -17254.665} C_VEL
LIN {X 0,Y 283.394,Z 421.056,A -85,B 0,C 180,E1 -17256.971,E2 -17256.971} C_VEL
LIN {X 0,Y 282.054,Z 425.115,A -85,B 0,C 180,E1 -17257.788,E2 -17257.788} C_VEL
LIN {X 0,Y 280.309,Z 435.623,A -85,B 0,C 180,E1 -17260.216,E2 -17260.216} C_VEL
LIN {X 0,Y 278.734,Z 446.077,A -85,B 0,C 180,E1 -17263.07,E2 -17263.07} C_VEL
LIN {X 0,Y 277.625,Z 454.237,A -85,B 0,C 180,E1 -17265.711,E2 -17265.711} C_VEL
LIN {X 0,Y 276.653,Z 462.638,A -85,B 0,C 180,E1 -17269.016,E2 -17269.016} C_VEL
LIN {X 0,Y 276.175,Z 468.647,A -85,B 0,C 180,E1 -17271.954,E2 -17271.954} C_VEL
LIN {X 0,Y 275.88,Z 473.355,A -85,B 0,C 180,E1 -17274.884,E2 -17274.884} C_VEL
LIN {X 0,Y 275.827,Z 476.166,A -85,B 0,C 180,E1 -17277.079,E2 -17277.079} C_VEL
LIN {X 0,Y 275.891,Z 478.922,A -85,B 0,C 180,E1 -17280,E2 -17280} C_VEL
LIN {X 0,Y 276.273,Z 480.691,A -85,B 0,C 180,E1 -17282.916,E2 -17282.916} C_VEL
LIN {X 0,Y 276.7,Z 481.381,A -85,B 0,C 180,E1 -17285.831,E2 -17285.831} C_VEL
LIN {X 0,Y 277.747,Z 480.964,A -85,B 0,C 180,E1 -17289.3,E2 -17289.3} C_VEL
LIN {X 0,Y 278.838,Z 479.892,A -85,B 0,C 180,E1 -17291.633,E2 -17291.633} C_VEL
LIN {X 0,Y 280.53,Z 477.722,A -85,B 0,C 180,E1 -17294.508,E2 -17294.508} C_VEL
LIN {X 0,Y 282.686,Z 474.545,A -85,B 0,C 180,E1 -17297.358,E2 -17297.358} C_VEL
LIN {X 0,Y 285.544,Z 470.355,A -85,B 0,C 180,E1 -17300.156,E2 -17300.156} C_VEL
LIN {X 0,Y 288.99,Z 465.151,A -85,B 0,C 180,E1 -17302.899,E2 -17302.899} C_VEL
LIN {X 0,Y 294.092,Z 457.098,A -85,B 0,C 180,E1 -17306.238,E2 -17306.238} C_VEL
LIN {X 0,Y 300.226,Z 447.137,A -85,B 0,C 180,E1 -17309.445,E2 -17309.445} C_VEL
LIN {X 0,Y 305.798,Z 437.754,A -85,B 0,C 180,E1 -17311.911,E2 -17311.911} C_VEL
LIN {X 0,Y 312.085,Z 426.836,A -85,B 0,C 180,E1 -17314.262,E2 -17314.262} C_VEL
LIN {X 0,Y 318.906,Z 414.4,A -85,B 0,C 180,E1 -17316.514,E2 -17316.514} C_VEL
LIN {X 0,Y 326.509,Z 399.989,A -85,B 0,C 180,E1 -17318.624,E2 -17318.624} C_VEL
LIN {X 0,Y 333.604,Z 385.652,A -85,B 0,C 180,E1 -17320.327,E2 -17320.327} C_VEL
LIN {X 0,Y 340.354,Z 370.947,A -85,B 0,C 180,E1 -17321.754,E2 -17321.754} C_VEL
LIN {X 0,Y 346.751,Z 355.682,A -85,B 0,C 180,E1 -17322.962,E2 -17322.962} C_VEL
LIN {X 0,Y 352.86,Z 339.221,A -85,B 0,C 180,E1 -17323.996,E2 -17323.996} C_VEL
LIN {X 0,Y 354.511,Z 334.242,A -85,B 0,C 180,E1 -17324.263,E2 -17324.263} C_VEL
LIN {X 0,Y 354.488,Z 334.374,A -85,B 0,C 180,E1 -17324.46,E2 -17324.46} C_VEL
LIN {X 0,Y 348.277,Z 352.643,A -85,B 0,C 180,E1 -17325.234,E2 -17325.234} C_VEL
LIN {X 0,Y 340.637,Z 372.131,A -85,B 0,C 180,E1 -17326.277,E2 -17326.277} C_VEL
LIN {X 0,Y 332.895,Z 389.913,A -85,B 0,C 180,E1 -17327.5,E2 -17327.5} C_VEL
LIN {X 0,Y 326.359,Z 404.049,A -85,B 0,C 180,E1 -17328.738,E2 -17328.738} C_VEL
LIN {X 0,Y 318.146,Z 421.007,A -85,B 0,C 180,E1 -17330.572,E2 -17330.572} C_VEL
LIN {X 0,Y 311.238,Z 434.975,A -85,B 0,C 180,E1 -17332.433,E2 -17332.433} C_VEL
LIN {X 0,Y 304.09,Z 449.111,A -85,B 0,C 180,E1 -17334.704,E2 -17334.704} C_VEL
LIN {X 0,Y 297.126,Z 463.039,A -85,B 0,C 180,E1 -17337.444,E2 -17337.444} C_VEL
LIN {X 0,Y 291.446,Z 474.683,A -85,B 0,C 180,E1 -17340.239,E2 -17340.239} C_VEL
LIN {X 0,Y 286.833,Z 484.472,A -85,B 0,C 180,E1 -17343.044,E2 -17343.044} C_VEL
LIN {X 0,Y 283.207,Z 492.685,A -85,B 0,C 180,E1 -17345.828,E2 -17345.828} C_VEL
LIN {X 0,Y 279.764,Z 501.286,A -85,B 0,C 180,E1 -17349.408,E2 -17349.408} C_VEL
LIN {X 0,Y 277.363,Z 508.191,A -85,B 0,C 180,E1 -17353.058,E2 -17353.058} C_VEL
LIN {X 0,Y 276.499,Z 511.578,A -85,B 0,C 180,E1 -17355.274,E2 -17355.274} C_VEL
LIN {X 0,Y 275.659,Z 515.113,A -85,B 0,C 180,E1 -17358.23,E2 -17358.23} C_VEL
LIN {X 0,Y 275.448,Z 517.724,A -85,B 0,C 180,E1 -17361.193,E2 -17361.193} C_VEL
LIN {X 0,Y 275.617,Z 519.201,A -85,B 0,C 180,E1 -17364.145,E2 -17364.145} C_VEL
LIN {X 0,Y 275.764,Z 519.675,A -85,B 0,C 180,E1 -17367.077,E2 -17367.077} C_VEL
LIN {X 0,Y 276.13,Z 518.941,A -85,B 0,C 180,E1 -17369.999,E2 -17369.999} C_VEL
LIN {X 0,Y 275.999,Z 517.057,A -85,B 0,C 180,E1 -17372.918,E2 -17372.918} C_VEL
LIN {X 0,Y 275.917,Z 513.891,A -85,B 0,C 180,E1 -17375.847,E2 -17375.847} C_VEL
LIN {X 0,Y 275.845,Z 510.701,A -85,B 0,C 180,E1 -17378.054,E2 -17378.054} C_VEL
LIN {X 0,Y 275.882,Z 505.163,A -85,B 0,C 180,E1 -17381.014,E2 -17381.014} C_VEL
LIN {X 0,Y 276.345,Z 498.206,A -85,B 0,C 180,E1 -17383.98,E2 -17383.98} C_VEL
LIN {X 0,Y 277.166,Z 489.64,A -85,B 0,C 180,E1 -17386.953,E2 -17386.953} C_VEL
LIN {X 0,Y 278.243,Z 480.686,A -85,B 0,C 180,E1 -17389.552,E2 -17389.552} C_VEL
LIN {X 0,Y 279.835,Z 470.126,A -85,B 0,C 180,E1 -17392.13,E2 -17392.13} C_VEL
LIN {X 0,Y 281.831,Z 457.666,A -85,B 0,C 180,E1 -17394.688,E2 -17394.688} C_VEL
LIN {X 0,Y 283.958,Z 444.9,A -85,B 0,C 180,E1 -17396.894,E2 -17396.894} C_VEL
LIN {X 0,Y 286.432,Z 430.504,A -85,B 0,C 180,E1 -17398.985,E2 -17398.985} C_VEL
LIN {X 0,Y 288.803,Z 416.114,A -85,B 0,C 180,E1 -17400.732,E2 -17400.732} C_VEL
LIN {X 0,Y 291.223,Z 400.743,A -85,B 0,C 180,E1 -17402.28,E2 -17402.28} C_VEL
LIN {X 0,Y 293.498,Z 384.375,A -85,B 0,C 180,E1 -17403.623,E2 -17403.623} C_VEL
LIN {X 0,Y 295.639,Z 367.025,A -85,B 0,C 180,E1 -17404.734,E2 -17404.734} C_VEL
LIN {X 0,Y 297.356,Z 350.405,A -85,B 0,C 180,E1 -17405.539,E2 -17405.539} C_VEL
LIN {X 0,Y 307.824,Z 203.128,A -85,B 0,C 180,E1 -17410.579,E2 -17410.579} C_VEL
LIN {X 0,Y 306.62,Z 192.119,A -85,B 0,C 180,E1 -17411.147,E2 -17411.147} C_VEL
LIN {X 0,Y 293.215,Z 161.577,A -85,B 0,C 180,E1 -17413.9,E2 -17413.9} C_VEL
LIN {X 0,Y 283.382,Z 140.444,A -85,B 0,C 180,E1 -17416.076,E2 -17416.076} C_VEL
LIN {X 0,Y 277.266,Z 122.261,A -85,B 0,C 180,E1 -17420.185,E2 -17420.185} C_VEL
LIN {X 0,Y 277.299,Z 122.257,A -85,B 0,C 180,E1 -17424.344,E2 -17424.344} C_VEL
LIN {X 0,Y 277.242,Z 122.264,A -85,B 0,C 180,E1 -17427.836,E2 -17427.836} C_VEL
LIN {X 0,Y 277.267,Z 122.259,A -85,B 0,C 180,E1 -17431.21,E2 -17431.21} C_VEL
LIN {X 0,Y 277.309,Z 122.257,A -85,B 0,C 180,E1 -17434.479,E2 -17434.479} C_VEL
LIN {X 0,Y 277.281,Z 122.26,A -85,B 0,C 180,E1 -17437.655,E2 -17437.655} C_VEL
LIN {X 0,Y 277.341,Z 122.25,A -85,B 0,C 180,E1 -17440.766,E2 -17440.766} C_VEL
LIN {X 0,Y 277.431,Z 122.238,A -85,B 0,C 180,E1 -17445.326,E2 -17445.326} C_VEL
LIN {X 0,Y 277.503,Z 122.231,A -85,B 0,C 180,E1 -17449.789,E2 -17449.789} C_VEL
LIN {X 0,Y 277.649,Z 122.21,A -85,B 0,C 180,E1 -17452.729,E2 -17452.729} C_VEL
LIN {X 0,Y 277.817,Z 122.189,A -85,B 0,C 180,E1 -17458.551,E2 -17458.551} C_VEL
LIN {X 0,Y 277.817,Z 122.191,A -85,B 0,C 180,E1 -17461.45,E2 -17461.45} C_VEL
LIN {X 0,Y 277.65,Z 122.211,A -85,B 0,C 180,E1 -17467.271,E2 -17467.271} C_VEL
LIN {X 0,Y 277.502,Z 122.228,A -85,B 0,C 180,E1 -17470.212,E2 -17470.212} C_VEL
LIN {X 0,Y 277.43,Z 122.238,A -85,B 0,C 180,E1 -17474.674,E2 -17474.674} C_VEL
LIN {X 0,Y 277.341,Z 122.251,A -85,B 0,C 180,E1 -17479.234,E2 -17479.234} C_VEL
LIN {X 0,Y 277.315,Z 122.248,A -85,B 0,C 180,E1 -17484.171,E2 -17484.171} C_VEL
LIN {X 0,Y 277.319,Z 122.253,A -85,B 0,C 180,E1 -17487.505,E2 -17487.505} C_VEL
LIN {X 0,Y 277.268,Z 122.256,A -85,B 0,C 180,E1 -17490.482,E2 -17490.482} C_VEL
LIN {X 0,Y 277.243,Z 122.26,A -85,B 0,C 180,E1 -17493.896,E2 -17493.896} C_VEL
LIN {X 0,Y 277.261,Z 122.257,A -85,B 0,C 180,E1 -17497.47,E2 -17497.47} C_VEL
LIN {X 0,Y 277.206,Z 122.267,A -85,B 0,C 180,E1 -17501.237,E2 -17501.237} C_VEL
LIN {X 0,Y 277.22,Z 122.262,A -85,B 0,C 180,E1 -17505.222,E2 -17505.222} C_VEL
LIN {X 0,Y 277.284,Z 122.255,A -85,B 0,C 180,E1 -17509.497,E2 -17509.497} C_VEL
LIN {X 0,Y 277.283,Z 122.258,A -85,B 0,C 180,E1 -17512.534,E2 -17512.534} C_VEL
LIN {X 0,Y 277.252,Z 122.259,A -85,B 0,C 180,E1 -17516.106,E2 -17516.106} C_VEL
LIN {X 0,Y 277.259,Z 122.258,A -85,B 0,C 180,E1 -17519.54,E2 -17519.54} C_VEL
LIN {X 0,Y 277.354,Z 122.248,A -85,B 0,C 180,E1 -17522.865,E2 -17522.865} C_VEL
LIN {X 0,Y 277.327,Z 122.252,A -85,B 0,C 180,E1 -17526.081,E2 -17526.081} C_VEL
LIN {X 0,Y 277.346,Z 122.25,A -85,B 0,C 180,E1 -17530.767,E2 -17530.767} C_VEL
LIN {X 0,Y 277.434,Z 122.233,A -85,B 0,C 180,E1 -17535.327,E2 -17535.327} C_VEL
LIN {X 0,Y 277.507,Z 122.229,A -85,B 0,C 180,E1 -17539.79,E2 -17539.79} C_VEL
LIN {X 0,Y 277.654,Z 122.21,A -85,B 0,C 180,E1 -17542.73,E2 -17542.73} C_VEL
LIN {X 0,Y 277.821,Z 122.19,A -85,B 0,C 180,E1 -17548.551,E2 -17548.551} C_VEL
LIN {X 0,Y 277.821,Z 122.188,A -85,B 0,C 180,E1 -17551.451,E2 -17551.451} C_VEL
LIN {X 0,Y 277.655,Z 122.21,A -85,B 0,C 180,E1 -17557.272,E2 -17557.272} C_VEL
LIN {X 0,Y 277.508,Z 122.227,A -85,B 0,C 180,E1 -17560.212,E2 -17560.212} C_VEL
LIN {X 0,Y 277.437,Z 122.238,A -85,B 0,C 180,E1 -17564.675,E2 -17564.675} C_VEL
LIN {X 0,Y 277.347,Z 122.246,A -85,B 0,C 180,E1 -17569.235,E2 -17569.235} C_VEL
LIN {X 0,Y 277.331,Z 122.252,A -85,B 0,C 180,E1 -17573.921,E2 -17573.921} C_VEL
LIN {X 0,Y 277.326,Z 122.252,A -85,B 0,C 180,E1 -17577.505,E2 -17577.505} C_VEL
LIN {X 0,Y 277.275,Z 122.258,A -85,B 0,C 180,E1 -17580.482,E2 -17580.482} C_VEL
LIN {X 0,Y 277.257,Z 122.261,A -85,B 0,C 180,E1 -17583.895,E2 -17583.895} C_VEL
LIN {X 0,Y 277.285,Z 122.257,A -85,B 0,C 180,E1 -17587.468,E2 -17587.468} C_VEL
LIN {X 0,Y 277.213,Z 122.268,A -85,B 0,C 180,E1 -17591.237,E2 -17591.237} C_VEL
LIN {X 0,Y 277.236,Z 122.264,A -85,B 0,C 180,E1 -17594.612,E2 -17594.612} C_VEL
LIN {X 0,Y 278.198,Z 125.06,A -85,B 0,C 180,E1 -17594.881,E2 -17594.881} C_VEL
LIN {X 0,Y 289.558,Z 146.391,A -85,B 0,C 180,E1 -17597.255,E2 -17597.255} C_VEL
LIN {X 0,Y 303.178,Z 173.568,A -85,B 0,C 180,E1 -17599.906,E2 -17599.906} C_VEL
LIN {X 0,Y 306.409,Z 180.244,A -85,B 0,C 180,E1 -17600.505,E2 -17600.505} C_VEL
LIN {X 0,Y 297.62,Z 306.604,A -85,B 0,C 180,E1 -17604.807,E2 -17604.807} C_VEL
LIN {X 0,Y 296.132,Z 324.776,A -85,B 0,C 180,E1 -17605.721,E2 -17605.721} C_VEL
LIN {X 0,Y 294.384,Z 342.397,A -85,B 0,C 180,E1 -17606.899,E2 -17606.899} C_VEL
LIN {X 0,Y 292.378,Z 358.813,A -85,B 0,C 180,E1 -17608.277,E2 -17608.277} C_VEL
LIN {X 0,Y 290.015,Z 375.649,A -85,B 0,C 180,E1 -17610.012,E2 -17610.012} C_VEL
LIN {X 0,Y 287.517,Z 391.858,A -85,B 0,C 180,E1 -17612.055,E2 -17612.055} C_VEL
LIN {X 0,Y 285.14,Z 406.35,A -85,B 0,C 180,E1 -17614.252,E2 -17614.252} C_VEL
LIN {X 0,Y 282.937,Z 419.267,A -85,B 0,C 180,E1 -17616.582,E2 -17616.582} C_VEL
LIN {X 0,Y 282.054,Z 425.115,A -85,B 0,C 180,E1 -17617.788,E2 -17617.788} C_VEL
LIN {X 0,Y 280.704,Z 429.138,A -85,B 0,C 180,E1 -17618.627,E2 -17618.627} C_VEL
LIN {X 0,Y 276.827,Z 435.421,A -85,B 0,C 180,E1 -17619.993,E2 -17619.993} C_VEL
LIN {X 0,Y 273.058,Z 441.321,A -85,B 0,C 180,E1 -17621.461,E2 -17621.461} C_VEL
LIN {X 0,Y 271.9,Z 444.744,A -85,B 0,C 180,E1 -17622.446,E2 -17622.446} C_VEL
LIN {X 0,Y 270.641,Z 453.71,A -85,B 0,C 180,E1 -17625.334,E2 -17625.334} C_VEL
LIN {X 0,Y 269.617,Z 462.346,A -85,B 0,C 180,E1 -17628.726,E2 -17628.726} C_VEL
LIN {X 0,Y 269.112,Z 468.493,A -85,B 0,C 180,E1 -17631.742,E2 -17631.742} C_VEL
LIN {X 0,Y 268.807,Z 473.406,A -85,B 0,C 180,E1 -17634.749,E2 -17634.749} C_VEL
LIN {X 0,Y 268.742,Z 476.323,A -85,B 0,C 180,E1 -17637.002,E2 -17637.002} C_VEL
LIN {X 0,Y 268.8,Z 479.274,A -85,B 0,C 180,E1 -17640,E2 -17640} C_VEL
LIN {X 0,Y 269.209,Z 481.156,A -85,B 0,C 180,E1 -17642.993,E2 -17642.993} C_VEL
LIN {X 0,Y 269.649,Z 482.052,A -85,B 0,C 180,E1 -17645.984,E2 -17645.984} C_VEL
LIN {X 0,Y 270.532,Z 481.989,A -85,B 0,C 180,E1 -17648.967,E2 -17648.967} C_VEL
LIN {X 0,Y 271.949,Z 480.907,A -85,B 0,C 180,E1 -17651.931,E2 -17651.931} C_VEL
LIN {X 0,Y 273.759,Z 478.942,A -85,B 0,C 180,E1 -17654.875,E2 -17654.875} C_VEL
LIN {X 0,Y 276.047,Z 475.958,A -85,B 0,C 180,E1 -17657.789,E2 -17657.789} C_VEL
LIN {X 0,Y 279.1,Z 472.043,A -85,B 0,C 180,E1 -17660.642,E2 -17660.642} C_VEL
LIN {X 0,Y 283.724,Z 465.682,A -85,B 0,C 180,E1 -17664.124,E2 -17664.124} C_VEL
LIN {X 0,Y 289.312,Z 457.642,A -85,B 0,C 180,E1 -17667.487,E2 -17667.487} C_VEL
LIN {X 0,Y 295.221,Z 448.877,A -85,B 0,C 180,E1 -17670.389,E2 -17670.389} C_VEL
LIN {X 0,Y 301.775,Z 438.788,A -85,B 0,C 180,E1 -17673.101,E2 -17673.101} C_VEL
LIN {X 0,Y 308.672,Z 427.822,A -85,B 0,C 180,E1 -17675.492,E2 -17675.492} C_VEL
LIN {X 0,Y 316.919,Z 414.021,A -85,B 0,C 180,E1 -17677.98,E2 -17677.98} C_VEL
LIN {X 0,Y 326.088,Z 397.784,A -85,B 0,C 180,E1 -17680.284,E2 -17680.284} C_VEL
LIN {X 0,Y 334.492,Z 381.859,A -85,B 0,C 180,E1 -17682.045,E2 -17682.045} C_VEL
LIN {X 0,Y 341.605,Z 367.142,A -85,B 0,C 180,E1 -17683.364,E2 -17683.364} C_VEL
LIN {X 0,Y 345.931,Z 357.459,A -85,B 0,C 180,E1 -17684.093,E2 -17684.093} C_VEL
LIN {X 0,Y 345.713,Z 358.045,A -85,B 0,C 180,E1 -17684.295,E2 -17684.295} C_VEL
LIN {X 0,Y 338.204,Z 375.431,A -85,B 0,C 180,E1 -17685.256,E2 -17685.256} C_VEL
LIN {X 0,Y 330.165,Z 392.299,A -85,B 0,C 180,E1 -17686.437,E2 -17686.437} C_VEL
LIN {X 0,Y 322.775,Z 406.84,A -85,B 0,C 180,E1 -17687.757,E2 -17687.757} C_VEL
LIN {X 0,Y 314.225,Z 422.971,A -85,B 0,C 180,E1 -17689.562,E2 -17689.562} C_VEL
LIN {X 0,Y 306.014,Z 438.091,A -85,B 0,C 180,E1 -17691.676,E2 -17691.676} C_VEL
LIN {X 0,Y 298.609,Z 451.51,A -85,B 0,C 180,E1 -17693.956,E2 -17693.956} C_VEL
LIN {X 0,Y 291.354,Z 464.792,A -85,B 0,C 180,E1 -17696.716,E2 -17696.716} C_VEL
LIN {X 0,Y 285.541,Z 475.763,A -85,B 0,C 180,E1 -17699.48,E2 -17699.48} C_VEL
LIN {X 0,Y 280.552,Z 485.395,A -85,B 0,C 180,E1 -17702.39,E2 -17702.39} C_VEL
LIN {X 0,Y 276.709,Z 493.225,A -85,B 0,C 180,E1 -17705.223,E2 -17705.223} C_VEL
LIN {X 0,Y 273.032,Z 501.515,A -85,B 0,C 180,E1 -17708.876,E2 -17708.876} C_VEL
LIN {X 0,Y 270.912,Z 506.97,A -85,B 0,C 180,E1 -17711.861,E2 -17711.861} C_VEL
LIN {X 0,Y 269.537,Z 511.402,A -85,B 0,C 180,E1 -17714.885,E2 -17714.885} C_VEL
LIN {X 0,Y 268.612,Z 514.822,A -85,B 0,C 180,E1 -17717.917,E2 -17717.917} C_VEL
LIN {X 0,Y 268.362,Z 517.243,A -85,B 0,C 180,E1 -17720.959,E2 -17720.959} C_VEL
LIN {X 0,Y 268.558,Z 518.63,A -85,B 0,C 180,E1 -17723.99,E2 -17723.99} C_VEL
LIN {X 0,Y 268.704,Z 518.935,A -85,B 0,C 180,E1 -17727,E2 -17727} C_VEL
LIN {X 0,Y 269.095,Z 518.125,A -85,B 0,C 180,E1 -17729.999,E2 -17729.999} C_VEL
LIN {X 0,Y 268.946,Z 516.064,A -85,B 0,C 180,E1 -17732.995,E2 -17732.995} C_VEL
LIN {X 0,Y 268.878,Z 512.817,A -85,B 0,C 180,E1 -17736,E2 -17736} C_VEL
LIN {X 0,Y 268.776,Z 508.15,A -85,B 0,C 180,E1 -17739.025,E2 -17739.025} C_VEL
LIN {X 0,Y 268.946,Z 502.113,A -85,B 0,C 180,E1 -17742.066,E2 -17742.066} C_VEL
LIN {X 0,Y 269.534,Z 494.593,A -85,B 0,C 180,E1 -17745.113,E2 -17745.113} C_VEL
LIN {X 0,Y 270.539,Z 485.378,A -85,B 0,C 180,E1 -17748.163,E2 -17748.163} C_VEL
LIN {X 0,Y 271.806,Z 475.713,A -85,B 0,C 180,E1 -17750.825,E2 -17750.825} C_VEL
LIN {X 0,Y 273.652,Z 464.374,A -85,B 0,C 180,E1 -17753.457,E2 -17753.457} C_VEL
LIN {X 0,Y 275.718,Z 452.001,A -85,B 0,C 180,E1 -17755.88,E2 -17755.88} C_VEL
LIN {X 0,Y 278.004,Z 438.573,A -85,B 0,C 180,E1 -17758.1,E2 -17758.1} C_VEL
LIN {X 0,Y 280.511,Z 424.326,A -85,B 0,C 180,E1 -17760.071,E2 -17760.071} C_VEL
LIN {X 0,Y 283.073,Z 408.93,A -85,B 0,C 180,E1 -17761.841,E2 -17761.841} C_VEL
LIN {X 0,Y 285.393,Z 393.608,A -85,B 0,C 180,E1 -17763.297,E2 -17763.297} C_VEL
LIN {X 0,Y 287.782,Z 376.489,A -85,B 0,C 180,E1 -17764.595,E2 -17764.595} C_VEL
LIN {X 0,Y 289.934,Z 358.71,A -85,B 0,C 180,E1 -17765.627,E2 -17765.627} C_VEL
LIN {X 0,Y 291.486,Z 340.048,A -85,B 0,C 180,E1 -17766.421,E2 -17766.421} C_VEL
LIN {X 0,Y 301.523,Z 204.105,A -85,B 0,C 180,E1 -17771.168,E2 -17771.168} C_VEL
LIN {X 0,Y 300.49,Z 194.567,A -85,B 0,C 180,E1 -17771.672,E2 -17771.672} C_VEL
LIN {X 0,Y 286.903,Z 163.646,A -85,B 0,C 180,E1 -17774.547,E2 -17774.547} C_VEL
LIN {X 0,Y 277.746,Z 144.027,A -85,B 0,C 180,E1 -17776.595,E2 -17776.595} C_VEL
LIN {X 0,Y 275.899,Z 139.999,A -85,B 0,C 180,E1 -17777.047,E2 -17777.047} C_VEL
LIN {X 0,Y 270.197,Z 123.141,A -85,B 0,C 180,E1 -17780.961,E2 -17780.961} C_VEL
LIN {X 0,Y 270.25,Z 123.134,A -85,B 0,C 180,E1 -17783.722,E2 -17783.722} C_VEL
LIN {X 0,Y 270.201,Z 123.139,A -85,B 0,C 180,E1 -17786.892,E2 -17786.892} C_VEL
LIN {X 0,Y 270.217,Z 123.139,A -85,B 0,C 180,E1 -17790.385,E2 -17790.385} C_VEL
LIN {X 0,Y 270.259,Z 123.134,A -85,B 0,C 180,E1 -17793.764,E2 -17793.764} C_VEL
LIN {X 0,Y 270.228,Z 123.137,A -85,B 0,C 180,E1 -17797.039,E2 -17797.039} C_VEL
LIN {X 0,Y 270.297,Z 123.13,A -85,B 0,C 180,E1 -17800.244,E2 -17800.244} C_VEL
LIN {X 0,Y 270.399,Z 123.114,A -85,B 0,C 180,E1 -17804.935,E2 -17804.935} C_VEL
LIN {X 0,Y 270.438,Z 123.108,A -85,B 0,C 180,E1 -17809.519,E2 -17809.519} C_VEL
LIN {X 0,Y 270.607,Z 123.087,A -85,B 0,C 180,E1 -17812.539,E2 -17812.539} C_VEL
LIN {X 0,Y 270.783,Z 123.066,A -85,B 0,C 180,E1 -17818.513,E2 -17818.513} C_VEL
LIN {X 0,Y 270.783,Z 123.067,A -85,B 0,C 180,E1 -17821.487,E2 -17821.487} C_VEL
LIN {X 0,Y 270.608,Z 123.09,A -85,B 0,C 180,E1 -17827.461,E2 -17827.461} C_VEL
LIN {X 0,Y 270.437,Z 123.107,A -85,B 0,C 180,E1 -17830.481,E2 -17830.481} C_VEL
LIN {X 0,Y 270.399,Z 123.116,A -85,B 0,C 180,E1 -17835.065,E2 -17835.065} C_VEL
LIN {X 0,Y 270.297,Z 123.127,A -85,B 0,C 180,E1 -17839.756,E2 -17839.756} C_VEL
LIN {X 0,Y 270.27,Z 123.126,A -85,B 0,C 180,E1 -17844.586,E2 -17844.586} C_VEL
LIN {X 0,Y 270.267,Z 123.13,A -85,B 0,C 180,E1 -17847.909,E2 -17847.909} C_VEL
LIN {X 0,Y 270.18,Z 123.14,A -85,B 0,C 180,E1 -17851.349,E2 -17851.349} C_VEL
LIN {X 0,Y 270.198,Z 123.142,A -85,B 0,C 180,E1 -17854.906,E2 -17854.906} C_VEL
LIN {X 0,Y 270.194,Z 123.138,A -85,B 0,C 180,E1 -17858.711,E2 -17858.711} C_VEL
LIN {X 0,Y 270.168,Z 123.143,A -85,B 0,C 180,E1 -17863.251,E2 -17863.251} C_VEL
LIN {X 0,Y 270.192,Z 123.137,A -85,B 0,C 180,E1 -17867.447,E2 -17867.447} C_VEL
LIN {X 0,Y 270.242,Z 123.132,A -85,B 0,C 180,E1 -17871.382,E2 -17871.382} C_VEL
LIN {X 0,Y 270.213,Z 123.136,A -85,B 0,C 180,E1 -17875.097,E2 -17875.097} C_VEL
LIN {X 0,Y 270.198,Z 123.138,A -85,B 0,C 180,E1 -17879.132,E2 -17879.132} C_VEL
LIN {X 0,Y 270.261,Z 123.128,A -85,B 0,C 180,E1 -17882.147,E2 -17882.147} C_VEL
LIN {X 0,Y 270.276,Z 123.129,A -85,B 0,C 180,E1 -17885.52,E2 -17885.52} C_VEL
LIN {X 0,Y 270.302,Z 123.126,A -85,B 0,C 180,E1 -17890.246,E2 -17890.246} C_VEL
LIN {X 0,Y 270.403,Z 123.11,A -85,B 0,C 180,E1 -17894.936,E2 -17894.936} C_VEL
LIN {X 0,Y 270.442,Z 123.108,A -85,B 0,C 180,E1 -17899.52,E2 -17899.52} C_VEL
LIN {X 0,Y 270.612,Z 123.089,A -85,B 0,C 180,E1 -17902.54,E2 -17902.54} C_VEL
LIN {X 0,Y 270.787,Z 123.067,A -85,B 0,C 180,E1 -17908.514,E2 -17908.514} C_VEL
LIN {X 0,Y 270.787,Z 123.065,A -85,B 0,C 180,E1 -17911.488,E2 -17911.488} C_VEL
LIN {X 0,Y 270.613,Z 123.089,A -85,B 0,C 180,E1 -17917.462,E2 -17917.462} C_VEL
LIN {X 0,Y 270.444,Z 123.105,A -85,B 0,C 180,E1 -17920.482,E2 -17920.482} C_VEL
LIN {X 0,Y 270.405,Z 123.114,A -85,B 0,C 180,E1 -17925.065,E2 -17925.065} C_VEL
LIN {X 0,Y 270.304,Z 123.128,A -85,B 0,C 180,E1 -17929.756,E2 -17929.756} C_VEL
LIN {X 0,Y 270.277,Z 123.129,A -85,B 0,C 180,E1 -17934.586,E2 -17934.586} C_VEL
LIN {X 0,Y 270.272,Z 123.131,A -85,B 0,C 180,E1 -17937.91,E2 -17937.91} C_VEL
LIN {X 0,Y 270.187,Z 123.142,A -85,B 0,C 180,E1 -17941.349,E2 -17941.349} C_VEL
LIN {X 0,Y 270.218,Z 123.137,A -85,B 0,C 180,E1 -17944.904,E2 -17944.904} C_VEL
LIN {X 0,Y 270.225,Z 123.136,A -85,B 0,C 180,E1 -17948.718,E2 -17948.718} C_VEL
LIN {X 0,Y 270.188,Z 123.144,A -85,B 0,C 180,E1 -17953.46,E2 -17953.46} C_VEL
LIN {X 0,Y 270.219,Z 123.282,A -85,B 0,C 180,E1 -17953.745,E2 -17953.745} C_VEL
LIN {X 0,Y 271.286,Z 126.122,A -85,B 0,C 180,E1 -17954.028,E2 -17954.028} C_VEL
LIN {X 0,Y 283.814,Z 149.725,A -85,B 0,C 180,E1 -17956.735,E2 -17956.735} C_VEL
LIN {X 0,Y 296.474,Z 175.112,A -85,B 0,C 180,E1 -17959.274,E2 -17959.274} C_VEL
LIN {X 0,Y 299.992,Z 182.374,A -85,B 0,C 180,E1 -17959.945,E2 -17959.945} C_VEL
LIN {X 0,Y 291.01,Z 307.018,A -85,B 0,C 180,E1 -17964.311,E2 -17964.311} C_VEL
LIN {X 0,Y 289.525,Z 324.711,A -85,B 0,C 180,E1 -17965.219,E2 -17965.219} C_VEL
LIN {X 0,Y 287.681,Z 342.704,A -85,B 0,C 180,E1 -17966.446,E2 -17966.446} C_VEL
LIN {X 0,Y 285.615,Z 359.092,A -85,B 0,C 180,E1 -17967.851,E2 -17967.851} C_VEL
LIN {X 0,Y 283.207,Z 375.953,A -85,B 0,C 180,E1 -17969.627,E2 -17969.627} C_VEL
LIN {X 0,Y 280.771,Z 391.385,A -85,B 0,C 180,E1 -17971.602,E2 -17971.602} C_VEL
LIN {X 0,Y 278.197,Z 406.704,A -85,B 0,C 180,E1 -17973.964,E2 -17973.964} C_VEL
LIN {X 0,Y 275.761,Z 420.707,A -85,B 0,C 180,E1 -17976.564,E2 -17976.564} C_VEL
LIN {X 0,Y 274.082,Z 431.569,A -85,B 0,C 180,E1 -17978.962,E2 -17978.962} C_VEL
LIN {X 0,Y 272.354,Z 441.681,A -85,B 0,C 180,E1 -17981.572,E2 -17981.572} C_VEL
LIN {X 0,Y 271.9,Z 444.744,A -85,B 0,C 180,E1 -17982.446,E2 -17982.446} C_VEL
LIN {X 0,Y 270.774,Z 448.109,A -85,B 0,C 180,E1 -17983.452,E2 -17983.452} C_VEL
LIN {X 0,Y 267.182,Z 453.242,A -85,B 0,C 180,E1 -17985.088,E2 -17985.088} C_VEL
LIN {X 0,Y 263.667,Z 458.055,A -85,B 0,C 180,E1 -17986.81,E2 -17986.81} C_VEL
LIN {X 0,Y 262.684,Z 460.791,A -85,B 0,C 180,E1 -17987.933,E2 -17987.933} C_VEL
LIN {X 0,Y 262.138,Z 466.875,A -85,B 0,C 180,E1 -17990.743,E2 -17990.743} C_VEL
LIN {X 0,Y 261.767,Z 472.249,A -85,B 0,C 180,E1 -17993.835,E2 -17993.835} C_VEL
LIN {X 0,Y 261.659,Z 476.45,A -85,B 0,C 180,E1 -17996.921,E2 -17996.921} C_VEL
LIN {X 0,Y 261.707,Z 479.597,A -85,B 0,C 180,E1 -18000,E2 -18000} C_VEL
LIN {X 0,Y 262.129,Z 481.61,A -85,B 0,C 180,E1 -18003.074,E2 -18003.074} C_VEL
LIN {X 0,Y 262.6,Z 482.727,A -85,B 0,C 180,E1 -18006.145,E2 -18006.145} C_VEL
LIN {X 0,Y 263.754,Z 482.738,A -85,B 0,C 180,E1 -18009.626,E2 -18009.626} C_VEL
LIN {X 0,Y 265.072,Z 481.941,A -85,B 0,C 180,E1 -18012.246,E2 -18012.246} C_VEL
LIN {X 0,Y 266.979,Z 480.12,A -85,B 0,C 180,E1 -18015.262,E2 -18015.262} C_VEL
LIN {X 0,Y 269.45,Z 477.405,A -85,B 0,C 180,E1 -18018.239,E2 -18018.239} C_VEL
LIN {X 0,Y 273.518,Z 472.624,A -85,B 0,C 180,E1 -18021.874,E2 -18021.874} C_VEL
LIN {X 0,Y 278.578,Z 466.307,A -85,B 0,C 180,E1 -18025.396,E2 -18025.396} C_VEL
LIN {X 0,Y 284.72,Z 458.328,A -85,B 0,C 180,E1 -18028.772,E2 -18028.772} C_VEL
LIN {X 0,Y 291.077,Z 449.707,A -85,B 0,C 180,E1 -18031.678,E2 -18031.678} C_VEL
LIN {X 0,Y 298.459,Z 439.306,A -85,B 0,C 180,E1 -18034.495,E2 -18034.495} C_VEL
LIN {X 0,Y 306.425,Z 427.661,A -85,B 0,C 180,E1 -18037.017,E2 -18037.017} C_VEL
LIN {X 0,Y 314.265,Z 415.626,A -85,B 0,C 180,E1 -18039.18,E2 -18039.18} C_VEL
LIN {X 0,Y 322.83,Z 401.782,A -85,B 0,C 180,E1 -18041.188,E2 -18041.188} C_VEL
LIN {X 0,Y 331.564,Z 386.694,A -85,B 0,C 180,E1 -18042.917,E2 -18042.917} C_VEL
LIN {X 0,Y 337.074,Z 376.497,A -85,B 0,C 180,E1 -18043.889,E2 -18043.889} C_VEL
LIN {X 0,Y 336.174,Z 378.389,A -85,B 0,C 180,E1 -18044.191,E2 -18044.191} C_VEL
LIN {X 0,Y 327.944,Z 394.238,A -85,B 0,C 180,E1 -18045.316,E2 -18045.316} C_VEL
LIN {X 0,Y 319.942,Z 408.778,A -85,B 0,C 180,E1 -18046.649,E2 -18046.649} C_VEL
LIN {X 0,Y 310.458,Z 425.189,A -85,B 0,C 180,E1 -18048.535,E2 -18048.535} C_VEL
LIN {X 0,Y 302.058,Z 439.359,A -85,B 0,C 180,E1 -18050.58,E2 -18050.58} C_VEL
LIN {X 0,Y 294.119,Z 452.496,A -85,B 0,C 180,E1 -18052.889,E2 -18052.889} C_VEL
LIN {X 0,Y 286.445,Z 465.3,A -85,B 0,C 180,E1 -18055.645,E2 -18055.645} C_VEL
LIN {X 0,Y 279.665,Z 476.877,A -85,B 0,C 180,E1 -18058.695,E2 -18058.695} C_VEL
LIN {X 0,Y 274.876,Z 485.348,A -85,B 0,C 180,E1 -18061.353,E2 -18061.353} C_VEL
LIN {X 0,Y 270.266,Z 493.846,A -85,B 0,C 180,E1 -18064.591,E2 -18064.591} C_VEL
LIN {X 0,Y 266.347,Z 501.785,A -85,B 0,C 180,E1 -18068.32,E2 -18068.32} C_VEL
LIN {X 0,Y 263.626,Z 508.163,A -85,B 0,C 180,E1 -18072.146,E2 -18072.146} C_VEL
LIN {X 0,Y 262.007,Z 513.011,A -85,B 0,C 180,E1 -18076.029,E2 -18076.029} C_VEL
LIN {X 0,Y 261.33,Z 515.765,A -85,B 0,C 180,E1 -18079.148,E2 -18079.148} C_VEL
LIN {X 0,Y 261.302,Z 517.535,A -85,B 0,C 180,E1 -18082.27,E2 -18082.27} C_VEL
LIN {X 0,Y 261.49,Z 518.093,A -85,B 0,C 180,E1 -18083.953,E2 -18083.953} C_VEL
LIN {X 0,Y 261.645,Z 518.182,A -85,B 0,C 180,E1 -18086.919,E2 -18086.919} C_VEL
LIN {X 0,Y 262.06,Z 517.295,A -85,B 0,C 180,E1 -18089.999,E2 -18089.999} C_VEL
LIN {X 0,Y 261.896,Z 515.054,A -85,B 0,C 180,E1 -18093.076,E2 -18093.076} C_VEL
LIN {X 0,Y 261.846,Z 511.641,A -85,B 0,C 180,E1 -18096.162,E2 -18096.162} C_VEL
LIN {X 0,Y 261.746,Z 508.148,A -85,B 0,C 180,E1 -18098.491,E2 -18098.491} C_VEL
LIN {X 0,Y 261.85,Z 502.312,A -85,B 0,C 180,E1 -18101.612,E2 -18101.612} C_VEL
LIN {X 0,Y 262.369,Z 494.993,A -85,B 0,C 180,E1 -18104.741,E2 -18104.741} C_VEL
LIN {X 0,Y 263.327,Z 485.958,A -85,B 0,C 180,E1 -18107.873,E2 -18107.873} C_VEL
LIN {X 0,Y 264.589,Z 476.485,A -85,B 0,C 180,E1 -18110.605,E2 -18110.605} C_VEL
LIN {X 0,Y 266.392,Z 465.383,A -85,B 0,C 180,E1 -18113.31,E2 -18113.31} C_VEL
LIN {X 0,Y 268.611,Z 452.261,A -85,B 0,C 180,E1 -18115.991,E2 -18115.991} C_VEL
LIN {X 0,Y 271.11,Z 437.965,A -85,B 0,C 180,E1 -18118.423,E2 -18118.423} C_VEL
LIN {X 0,Y 273.701,Z 423.487,A -85,B 0,C 180,E1 -18120.472,E2 -18120.472} C_VEL
LIN {X 0,Y 276.332,Z 408.069,A -85,B 0,C 180,E1 -18122.281,E2 -18122.281} C_VEL
LIN {X 0,Y 278.759,Z 392.405,A -85,B 0,C 180,E1 -18123.795,E2 -18123.795} C_VEL
LIN {X 0,Y 281.156,Z 375.602,A -85,B 0,C 180,E1 -18125.093,E2 -18125.093} C_VEL
LIN {X 0,Y 283.342,Z 357.835,A -85,B 0,C 180,E1 -18126.146,E2 -18126.146} C_VEL
LIN {X 0,Y 284.916,Z 339.236,A -85,B 0,C 180,E1 -18126.959,E2 -18126.959} C_VEL
LIN {X 0,Y 295.217,Z 204.929,A -85,B 0,C 180,E1 -18131.784,E2 -18131.784} C_VEL
LIN {X 0,Y 294.344,Z 197.046,A -85,B 0,C 180,E1 -18132.215,E2 -18132.215} C_VEL
LIN {X 0,Y 280.502,Z 165.394,A -85,B 0,C 180,E1 -18135.229,E2 -18135.229} C_VEL
LIN {X 0,Y 269.974,Z 142.871,A -85,B 0,C 180,E1 -18137.679,E2 -18137.679} C_VEL
LIN {X 0,Y 268.378,Z 139.366,A -85,B 0,C 180,E1 -18138.105,E2 -18138.105} C_VEL
LIN {X 0,Y 263.149,Z 124.019,A -85,B 0,C 180,E1 -18141.796,E2 -18141.796} C_VEL
LIN {X 0,Y 263.179,Z 124.016,A -85,B 0,C 180,E1 -18145.89,E2 -18145.89} C_VEL
LIN {X 0,Y 263.144,Z 124.019,A -85,B 0,C 180,E1 -18149.506,E2 -18149.506} C_VEL
LIN {X 0,Y 263.188,Z 124.014,A -85,B 0,C 180,E1 -18153.002,E2 -18153.002} C_VEL
LIN {X 0,Y 263.18,Z 124.017,A -85,B 0,C 180,E1 -18156.387,E2 -18156.387} C_VEL
LIN {X 0,Y 263.259,Z 124.005,A -85,B 0,C 180,E1 -18159.693,E2 -18159.693} C_VEL
LIN {X 0,Y 263.347,Z 123.993,A -85,B 0,C 180,E1 -18164.522,E2 -18164.522} C_VEL
LIN {X 0,Y 263.37,Z 123.987,A -85,B 0,C 180,E1 -18169.234,E2 -18169.234} C_VEL
LIN {X 0,Y 263.569,Z 123.965,A -85,B 0,C 180,E1 -18172.338,E2 -18172.338} C_VEL
LIN {X 0,Y 263.748,Z 123.942,A -85,B 0,C 180,E1 -18178.473,E2 -18178.473} C_VEL
LIN {X 0,Y 263.748,Z 123.944,A -85,B 0,C 180,E1 -18181.527,E2 -18181.527} C_VEL
LIN {X 0,Y 263.569,Z 123.967,A -85,B 0,C 180,E1 -18187.662,E2 -18187.662} C_VEL
LIN {X 0,Y 263.37,Z 123.988,A -85,B 0,C 180,E1 -18190.766,E2 -18190.766} C_VEL
LIN {X 0,Y 263.347,Z 123.994,A -85,B 0,C 180,E1 -18195.478,E2 -18195.478} C_VEL
LIN {X 0,Y 263.26,Z 124.002,A -85,B 0,C 180,E1 -18200.307,E2 -18200.307} C_VEL
LIN {X 0,Y 263.204,Z 124.011,A -85,B 0,C 180,E1 -18205.292,E2 -18205.292} C_VEL
LIN {X 0,Y 263.175,Z 124.015,A -85,B 0,C 180,E1 -18208.73,E2 -18208.73} C_VEL
LIN {X 0,Y 263.129,Z 124.016,A -85,B 0,C 180,E1 -18212.289,E2 -18212.289} C_VEL
LIN {X 0,Y 263.178,Z 124.015,A -85,B 0,C 180,E1 -18216.764,E2 -18216.764} C_VEL
LIN {X 0,Y 263.122,Z 124.02,A -85,B 0,C 180,E1 -18221.594,E2 -18221.594} C_VEL
LIN {X 0,Y 263.131,Z 124.015,A -85,B 0,C 180,E1 -18226.019,E2 -18226.019} C_VEL
LIN {X 0,Y 263.152,Z 124.016,A -85,B 0,C 180,E1 -18230.137,E2 -18230.137} C_VEL
LIN {X 0,Y 263.186,Z 124.008,A -85,B 0,C 180,E1 -18234.023,E2 -18234.023} C_VEL
LIN {X 0,Y 263.131,Z 124.018,A -85,B 0,C 180,E1 -18237.713,E2 -18237.713} C_VEL
LIN {X 0,Y 263.196,Z 124.006,A -85,B 0,C 180,E1 -18241.785,E2 -18241.785} C_VEL
LIN {X 0,Y 263.224,Z 124.007,A -85,B 0,C 180,E1 -18245.201,E2 -18245.201} C_VEL
LIN {X 0,Y 263.268,Z 123.999,A -85,B 0,C 180,E1 -18249.695,E2 -18249.695} C_VEL
LIN {X 0,Y 263.351,Z 123.99,A -85,B 0,C 180,E1 -18254.523,E2 -18254.523} C_VEL
LIN {X 0,Y 263.374,Z 123.988,A -85,B 0,C 180,E1 -18259.235,E2 -18259.235} C_VEL
LIN {X 0,Y 263.573,Z 123.966,A -85,B 0,C 180,E1 -18262.339,E2 -18262.339} C_VEL
LIN {X 0,Y 263.752,Z 123.943,A -85,B 0,C 180,E1 -18268.474,E2 -18268.474} C_VEL
LIN {X 0,Y 263.752,Z 123.941,A -85,B 0,C 180,E1 -18271.528,E2 -18271.528} C_VEL
LIN {X 0,Y 263.575,Z 123.967,A -85,B 0,C 180,E1 -18277.663,E2 -18277.663} C_VEL
LIN {X 0,Y 263.376,Z 123.985,A -85,B 0,C 180,E1 -18280.767,E2 -18280.767} C_VEL
LIN {X 0,Y 263.353,Z 123.995,A -85,B 0,C 180,E1 -18285.479,E2 -18285.479} C_VEL
LIN {X 0,Y 263.267,Z 124.003,A -85,B 0,C 180,E1 -18290.307,E2 -18290.307} C_VEL
LIN {X 0,Y 263.211,Z 124.011,A -85,B 0,C 180,E1 -18295.292,E2 -18295.292} C_VEL
LIN {X 0,Y 263.178,Z 124.014,A -85,B 0,C 180,E1 -18298.731,E2 -18298.731} C_VEL
LIN {X 0,Y 263.136,Z 124.02,A -85,B 0,C 180,E1 -18302.289,E2 -18302.289} C_VEL
LIN {X 0,Y 263.191,Z 124.014,A -85,B 0,C 180,E1 -18305.979,E2 -18305.979} C_VEL
LIN {X 0,Y 263.118,Z 124.02,A -85,B 0,C 180,E1 -18309.871,E2 -18309.871} C_VEL
LIN {X 0,Y 263.141,Z 124.018,A -85,B 0,C 180,E1 -18312.797,E2 -18312.797} C_VEL
LIN {X 0,Y 264.193,Z 126.908,A -85,B 0,C 180,E1 -18313.106,E2 -18313.106} C_VEL
LIN {X 0,Y 276.943,Z 150.887,A -85,B 0,C 180,E1 -18315.969,E2 -18315.969} C_VEL
LIN {X 0,Y 290.71,Z 178.439,A -85,B 0,C 180,E1 -18318.805,E2 -18318.805} C_VEL
LIN {X 0,Y 293.618,Z 184.873,A -85,B 0,C 180,E1 -18319.395,E2 -18319.395} C_VEL
LIN {X 0,Y 284.331,Z 307.974,A -85,B 0,C 180,E1 -18323.833,E2 -18323.833} C_VEL
LIN {X 0,Y 282.769,Z 326.189,A -85,B 0,C 180,E1 -18324.809,E2 -18324.809} C_VEL
LIN {X 0,Y 280.877,Z 343.757,A -85,B 0,C 180,E1 -18326.046,E2 -18326.046} C_VEL
LIN {X 0,Y 278.889,Z 359.254,A -85,B 0,C 180,E1 -18327.408,E2 -18327.408} C_VEL
LIN {X 0,Y 276.413,Z 376.173,A -85,B 0,C 180,E1 -18329.223,E2 -18329.223} C_VEL
LIN {X 0,Y 273.9,Z 391.627,A -85,B 0,C 180,E1 -18331.242,E2 -18331.242} C_VEL
LIN {X 0,Y 271.267,Z 406.996,A -85,B 0,C 180,E1 -18333.661,E2 -18333.661} C_VEL
LIN {X 0,Y 268.917,Z 420.264,A -85,B 0,C 180,E1 -18336.166,E2 -18336.166} C_VEL
LIN {X 0,Y 267.029,Z 431.925,A -85,B 0,C 180,E1 -18338.784,E2 -18338.784} C_VEL
LIN {X 0,Y 265.275,Z 442.086,A -85,B 0,C 180,E1 -18341.463,E2 -18341.463} C_VEL
LIN {X 0,Y 263.883,Z 451.937,A -85,B 0,C 180,E1 -18344.554,E2 -18344.554} C_VEL
LIN {X 0,Y 262.758,Z 460.116,A -85,B 0,C 180,E1 -18347.644,E2 -18347.644} C_VEL
LIN {X 0,Y 262.684,Z 460.791,A -85,B 0,C 180,E1 -18347.933,E2 -18347.933} C_VEL
LIN {X 0,Y 261.764,Z 463.438,A -85,B 0,C 180,E1 -18349.074,E2 -18349.074} C_VEL
LIN {X 0,Y 258.561,Z 467.377,A -85,B 0,C 180,E1 -18350.951,E2 -18350.951} C_VEL
LIN {X 0,Y 255.429,Z 470.943,A -85,B 0,C 180,E1 -18352.908,E2 -18352.908} C_VEL
LIN {X 0,Y 254.646,Z 472.91,A -85,B 0,C 180,E1 -18354.152,E2 -18354.152} C_VEL
LIN {X 0,Y 254.578,Z 476.565,A -85,B 0,C 180,E1 -18356.835,E2 -18356.835} C_VEL
LIN {X 0,Y 254.611,Z 479.825,A -85,B 0,C 180,E1 -18360,E2 -18360} C_VEL
LIN {X 0,Y 255.049,Z 482.053,A -85,B 0,C 180,E1 -18363.159,E2 -18363.159} C_VEL
LIN {X 0,Y 255.554,Z 483.323,A -85,B 0,C 180,E1 -18366.315,E2 -18366.315} C_VEL
LIN {X 0,Y 256.766,Z 483.547,A -85,B 0,C 180,E1 -18369.81,E2 -18369.81} C_VEL
LIN {X 0,Y 258.204,Z 482.934,A -85,B 0,C 180,E1 -18372.577,E2 -18372.577} C_VEL
LIN {X 0,Y 260.215,Z 481.324,A -85,B 0,C 180,E1 -18375.669,E2 -18375.669} C_VEL
LIN {X 0,Y 262.863,Z 478.844,A -85,B 0,C 180,E1 -18378.713,E2 -18378.713} C_VEL
LIN {X 0,Y 267.158,Z 474.356,A -85,B 0,C 180,E1 -18382.423,E2 -18382.423} C_VEL
LIN {X 0,Y 272.48,Z 468.394,A -85,B 0,C 180,E1 -18386.006,E2 -18386.006} C_VEL
LIN {X 0,Y 278.911,Z 460.857,A -85,B 0,C 180,E1 -18389.43,E2 -18389.43} C_VEL
LIN {X 0,Y 286.362,Z 451.69,A -85,B 0,C 180,E1 -18392.679,E2 -18392.679} C_VEL
LIN {X 0,Y 293.979,Z 441.913,A -85,B 0,C 180,E1 -18395.431,E2 -18395.431} C_VEL
LIN {X 0,Y 303.547,Z 429.158,A -85,B 0,C 180,E1 -18398.268,E2 -18398.268} C_VEL
LIN {X 0,Y 310.754,Z 418.986,A -85,B 0,C 180,E1 -18400.132,E2 -18400.132} C_VEL
LIN {X 0,Y 320.889,Z 404.087,A -85,B 0,C 180,E1 -18402.336,E2 -18402.336} C_VEL
LIN {X 0,Y 327.871,Z 393.056,A -85,B 0,C 180,E1 -18403.64,E2 -18403.64} C_VEL
LIN {X 0,Y 327.334,Z 394.111,A -85,B 0,C 180,E1 -18404.006,E2 -18404.006} C_VEL
LIN {X 0,Y 319.229,Z 407.759,A -85,B 0,C 180,E1 -18405.21,E2 -18405.21} C_VEL
LIN {X 0,Y 309.208,Z 423.813,A -85,B 0,C 180,E1 -18407.009,E2 -18407.009} C_VEL
LIN {X 0,Y 300.079,Z 437.985,A -85,B 0,C 180,E1 -18409.021,E2 -18409.021} C_VEL
LIN {X 0,Y 291.695,Z 450.667,A -85,B 0,C 180,E1 -18411.211,E2 -18411.211} C_VEL
LIN {X 0,Y 283.373,Z 463.337,A -85,B 0,C 180,E1 -18413.911,E2 -18413.911} C_VEL
LIN {X 0,Y 276.137,Z 474.528,A -85,B 0,C 180,E1 -18416.824,E2 -18416.824} C_VEL
LIN {X 0,Y 269.912,Z 484.365,A -85,B 0,C 180,E1 -18419.917,E2 -18419.917} C_VEL
LIN {X 0,Y 264.879,Z 492.772,A -85,B 0,C 180,E1 -18423.187,E2 -18423.187} C_VEL
LIN {X 0,Y 260.437,Z 500.678,A -85,B 0,C 180,E1 -18426.964,E2 -18426.964} C_VEL
LIN {X 0,Y 257.239,Z 507.076,A -85,B 0,C 180,E1 -18430.861,E2 -18430.861} C_VEL
LIN {X 0,Y 255.496,Z 511.452,A -85,B 0,C 180,E1 -18434.312,E2 -18434.312} C_VEL
LIN {X 0,Y 254.264,Z 515.396,A -85,B 0,C 180,E1 -18438.843,E2 -18438.843} C_VEL
LIN {X 0,Y 254.226,Z 516.96,A -85,B 0,C 180,E1 -18442.054,E2 -18442.054} C_VEL
LIN {X 0,Y 254.452,Z 517.581,A -85,B 0,C 180,E1 -18445.246,E2 -18445.246} C_VEL
LIN {X 0,Y 254.762,Z 517.02,A -85,B 0,C 180,E1 -18448.418,E2 -18448.418} C_VEL
LIN {X 0,Y 255.024,Z 516.362,A -85,B 0,C 180,E1 -18449.999,E2 -18449.999} C_VEL
LIN {X 0,Y 254.848,Z 514.027,A -85,B 0,C 180,E1 -18453.161,E2 -18453.161} C_VEL
LIN {X 0,Y 254.826,Z 509.714,A -85,B 0,C 180,E1 -18456.852,E2 -18456.852} C_VEL
LIN {X 0,Y 254.725,Z 503.97,A -85,B 0,C 180,E1 -18460.33,E2 -18460.33} C_VEL
LIN {X 0,Y 255.088,Z 497.198,A -85,B 0,C 180,E1 -18463.543,E2 -18463.543} C_VEL
LIN {X 0,Y 255.854,Z 488.818,A -85,B 0,C 180,E1 -18466.762,E2 -18466.762} C_VEL
LIN {X 0,Y 256.988,Z 480.012,A -85,B 0,C 180,E1 -18469.572,E2 -18469.572} C_VEL
LIN {X 0,Y 258.677,Z 468.967,A -85,B 0,C 180,E1 -18472.521,E2 -18472.521} C_VEL
LIN {X 0,Y 260.65,Z 457.34,A -85,B 0,C 180,E1 -18475.129,E2 -18475.129} C_VEL
LIN {X 0,Y 263.008,Z 444.137,A -85,B 0,C 180,E1 -18477.627,E2 -18477.627} C_VEL
LIN {X 0,Y 265.721,Z 429.433,A -85,B 0,C 180,E1 -18479.947,E2 -18479.947} C_VEL
LIN {X 0,Y 268.487,Z 413.615,A -85,B 0,C 180,E1 -18482.009,E2 -18482.009} C_VEL
LIN {X 0,Y 271.124,Z 397.934,A -85,B 0,C 180,E1 -18483.682,E2 -18483.682} C_VEL
LIN {X 0,Y 273.715,Z 380.521,A -85,B 0,C 180,E1 -18485.176,E2 -18485.176} C_VEL
LIN {X 0,Y 276.05,Z 362.829,A -85,B 0,C 180,E1 -18486.349,E2 -18486.349} C_VEL
LIN {X 0,Y 277.805,Z 345.494,A -85,B 0,C 180,E1 -18487.212,E2 -18487.212} C_VEL
LIN {X 0,Y 288.907,Z 205.92,A -85,B 0,C 180,E1 -18492.405,E2 -18492.405} C_VEL
LIN {X 0,Y 288.306,Z 199.69,A -85,B 0,C 180,E1 -18492.748,E2 -18492.748} C_VEL
LIN {X 0,Y 274.604,Z 168.302,A -85,B 0,C 180,E1 -18495.813,E2 -18495.813} C_VEL
LIN {X 0,Y 264.537,Z 146.723,A -85,B 0,C 180,E1 -18498.216,E2 -18498.216} C_VEL
LIN {X 0,Y 260.818,Z 138.752,A -85,B 0,C 180,E1 -18499.199,E2 -18499.199} C_VEL
LIN {X 0,Y 256.147,Z 124.891,A -85,B 0,C 180,E1 -18502.698,E2 -18502.698} C_VEL
LIN {X 0,Y 256.081,Z 124.898,A -85,B 0,C 180,E1 -18506.71,E2 -18506.71} C_VEL
LIN {X 0,Y 256.131,Z 124.893,A -85,B 0,C 180,E1 -18511.406,E2 -18511.406} C_VEL
LIN {X 0,Y 256.163,Z 124.893,A -85,B 0,C 180,E1 -18515.699,E2 -18515.699} C_VEL
LIN {X 0,Y 256.162,Z 124.888,A -85,B 0,C 180,E1 -18519.105,E2 -18519.105} C_VEL
LIN {X 0,Y 256.296,Z 124.874,A -85,B 0,C 180,E1 -18524.085,E2 -18524.085} C_VEL
LIN {X 0,Y 256.306,Z 124.866,A -85,B 0,C 180,E1 -18528.934,E2 -18528.934} C_VEL
LIN {X 0,Y 256.536,Z 124.842,A -85,B 0,C 180,E1 -18532.127,E2 -18532.127} C_VEL
LIN {X 0,Y 256.711,Z 124.819,A -85,B 0,C 180,E1 -18538.431,E2 -18538.431} C_VEL
LIN {X 0,Y 256.711,Z 124.82,A -85,B 0,C 180,E1 -18541.569,E2 -18541.569} C_VEL
LIN {X 0,Y 256.537,Z 124.842,A -85,B 0,C 180,E1 -18547.873,E2 -18547.873} C_VEL
LIN {X 0,Y 256.306,Z 124.869,A -85,B 0,C 180,E1 -18551.066,E2 -18551.066} C_VEL
LIN {X 0,Y 256.296,Z 124.869,A -85,B 0,C 180,E1 -18555.915,E2 -18555.915} C_VEL
LIN {X 0,Y 256.163,Z 124.888,A -85,B 0,C 180,E1 -18560.896,E2 -18560.896} C_VEL
LIN {X 0,Y 256.184,Z 124.883,A -85,B 0,C 180,E1 -18565.139,E2 -18565.139} C_VEL
LIN {X 0,Y 256.109,Z 124.892,A -85,B 0,C 180,E1 -18569.6,E2 -18569.6} C_VEL
LIN {X 0,Y 256.064,Z 124.901,A -85,B 0,C 180,E1 -18573.293,E2 -18573.293} C_VEL
LIN {X 0,Y 256.11,Z 124.892,A -85,B 0,C 180,E1 -18577.271,E2 -18577.271} C_VEL
LIN {X 0,Y 256.052,Z 124.902,A -85,B 0,C 180,E1 -18581.204,E2 -18581.204} C_VEL
LIN {X 0,Y 256.063,Z 124.895,A -85,B 0,C 180,E1 -18585.529,E2 -18585.529} C_VEL
LIN {X 0,Y 256.081,Z 124.899,A -85,B 0,C 180,E1 -18588.803,E2 -18588.803} C_VEL
LIN {X 0,Y 256.152,Z 124.886,A -85,B 0,C 180,E1 -18592.872,E2 -18592.872} C_VEL
LIN {X 0,Y 256.083,Z 124.9,A -85,B 0,C 180,E1 -18596.711,E2 -18596.711} C_VEL
LIN {X 0,Y 256.132,Z 124.885,A -85,B 0,C 180,E1 -18601.408,E2 -18601.408} C_VEL
LIN {X 0,Y 256.167,Z 124.886,A -85,B 0,C 180,E1 -18605.7,E2 -18605.7} C_VEL
LIN {X 0,Y 256.218,Z 124.877,A -85,B 0,C 180,E1 -18609.11,E2 -18609.11} C_VEL
LIN {X 0,Y 256.3,Z 124.872,A -85,B 0,C 180,E1 -18614.086,E2 -18614.086} C_VEL
LIN {X 0,Y 256.31,Z 124.869,A -85,B 0,C 180,E1 -18618.935,E2 -18618.935} C_VEL
LIN {X 0,Y 256.541,Z 124.84,A -85,B 0,C 180,E1 -18622.128,E2 -18622.128} C_VEL
LIN {X 0,Y 256.715,Z 124.82,A -85,B 0,C 180,E1 -18628.432,E2 -18628.432} C_VEL
LIN {X 0,Y 256.715,Z 124.818,A -85,B 0,C 180,E1 -18631.57,E2 -18631.57} C_VEL
LIN {X 0,Y 256.542,Z 124.845,A -85,B 0,C 180,E1 -18637.874,E2 -18637.874} C_VEL
LIN {X 0,Y 256.312,Z 124.865,A -85,B 0,C 180,E1 -18641.067,E2 -18641.067} C_VEL
LIN {X 0,Y 256.302,Z 124.872,A -85,B 0,C 180,E1 -18645.916,E2 -18645.916} C_VEL
LIN {X 0,Y 256.172,Z 124.886,A -85,B 0,C 180,E1 -18650.896,E2 -18650.896} C_VEL
LIN {X 0,Y 256.191,Z 124.885,A -85,B 0,C 180,E1 -18655.139,E2 -18655.139} C_VEL
LIN {X 0,Y 256.113,Z 124.899,A -85,B 0,C 180,E1 -18659.601,E2 -18659.601} C_VEL
LIN {X 0,Y 256.088,Z 124.901,A -85,B 0,C 180,E1 -18663.291,E2 -18663.291} C_VEL
LIN {X 0,Y 256.132,Z 124.892,A -85,B 0,C 180,E1 -18667.276,E2 -18667.276} C_VEL
LIN {X 0,Y 256.1,Z 124.897,A -85,B 0,C 180,E1 -18671.84,E2 -18671.84} C_VEL
LIN {X 0,Y 257.136,Z 127.797,A -85,B 0,C 180,E1 -18672.16,E2 -18672.16} C_VEL
LIN {X 0,Y 266.878,Z 145.932,A -85,B 0,C 180,E1 -18674.446,E2 -18674.446} C_VEL
LIN {X 0,Y 279.23,Z 170.257,A -85,B 0,C 180,E1 -18677.158,E2 -18677.158} C_VEL
LIN {X 0,Y 287.118,Z 186.443,A -85,B 0,C 180,E1 -18678.774,E2 -18678.774} C_VEL
LIN {X 0,Y 277.754,Z 307.854,A -85,B 0,C 180,E1 -18683.289,E2 -18683.289} C_VEL
LIN {X 0,Y 276.144,Z 326.058,A -85,B 0,C 180,E1 -18684.28,E2 -18684.28} C_VEL
LIN {X 0,Y 274.228,Z 343.456,A -85,B 0,C 180,E1 -18685.526,E2 -18685.526} C_VEL
LIN {X 0,Y 271.907,Z 361.122,A -85,B 0,C 180,E1 -18687.126,E2 -18687.126} C_VEL
LIN {X 0,Y 269.383,Z 377.665,A -85,B 0,C 180,E1 -18688.972,E2 -18688.972} C_VEL
LIN {X 0,Y 266.788,Z 393.056,A -85,B 0,C 180,E1 -18691.05,E2 -18691.05} C_VEL
LIN {X 0,Y 264.334,Z 407.211,A -85,B 0,C 180,E1 -18693.342,E2 -18693.342} C_VEL
LIN {X 0,Y 261.826,Z 420.957,A -85,B 0,C 180,E1 -18695.998,E2 -18695.998} C_VEL
LIN {X 0,Y 260.002,Z 432.231,A -85,B 0,C 180,E1 -18698.598,E2 -18698.598} C_VEL
LIN {X 0,Y 258.201,Z 442.435,A -85,B 0,C 180,E1 -18701.348,E2 -18701.348} C_VEL
LIN {X 0,Y 256.757,Z 452.332,A -85,B 0,C 180,E1 -18704.521,E2 -18704.521} C_VEL
LIN {X 0,Y 255.743,Z 459.65,A -85,B 0,C 180,E1 -18707.3,E2 -18707.3} C_VEL
LIN {X 0,Y 255.105,Z 466.553,A -85,B 0,C 180,E1 -18710.485,E2 -18710.485} C_VEL
LIN {X 0,Y 254.697,Z 472.143,A -85,B 0,C 180,E1 -18713.663,E2 -18713.663} C_VEL
LIN {X 0,Y 254.646,Z 472.91,A -85,B 0,C 180,E1 -18714.152,E2 -18714.152} C_VEL
LIN {X 0,Y 253.889,Z 474.779,A -85,B 0,C 180,E1 -18715.403,E2 -18715.403} C_VEL
LIN {X 0,Y 250.949,Z 477.434,A -85,B 0,C 180,E1 -18717.468,E2 -18717.468} C_VEL
LIN {X 0,Y 248.563,Z 479.257,A -85,B 0,C 180,E1 -18719.17,E2 -18719.17} C_VEL
LIN {X 0,Y 247.633,Z 480.476,A -85,B 0,C 180,E1 -18720.499,E2 -18720.499} C_VEL
LIN {X 0,Y 247.605,Z 480.817,A -85,B 0,C 180,E1 -18720.95,E2 -18720.95} C_VEL
LIN {X 0,Y 247.969,Z 482.489,A -85,B 0,C 180,E1 -18723.249,E2 -18723.249} C_VEL
LIN {X 0,Y 248.515,Z 483.881,A -85,B 0,C 180,E1 -18726.495,E2 -18726.495} C_VEL
LIN {X 0,Y 249.782,Z 484.365,A -85,B 0,C 180,E1 -18730.004,E2 -18730.004} C_VEL
LIN {X 0,Y 251.328,Z 483.883,A -85,B 0,C 180,E1 -18732.927,E2 -18732.927} C_VEL
LIN {X 0,Y 253.484,Z 482.549,A -85,B 0,C 180,E1 -18736.096,E2 -18736.096} C_VEL
LIN {X 0,Y 256.287,Z 480.236,A -85,B 0,C 180,E1 -18739.212,E2 -18739.212} C_VEL
LIN {X 0,Y 259.841,Z 477.064,A -85,B 0,C 180,E1 -18742.251,E2 -18742.251} C_VEL
LIN {X 0,Y 265.27,Z 471.764,A -85,B 0,C 180,E1 -18745.922,E2 -18745.922} C_VEL
LIN {X 0,Y 271.717,Z 464.99,A -85,B 0,C 180,E1 -18749.435,E2 -18749.435} C_VEL
LIN {X 0,Y 279.304,Z 456.642,A -85,B 0,C 180,E1 -18752.751,E2 -18752.751} C_VEL
LIN {X 0,Y 287.978,Z 446.638,A -85,B 0,C 180,E1 -18755.853,E2 -18755.853} C_VEL
LIN {X 0,Y 296.773,Z 436.068,A -85,B 0,C 180,E1 -18758.435,E2 -18758.435} C_VEL
LIN {X 0,Y 306.271,Z 424.016,A -85,B 0,C 180,E1 -18760.843,E2 -18760.843} C_VEL
LIN {X 0,Y 316.706,Z 410.055,A -85,B 0,C 180,E1 -18763.029,E2 -18763.029} C_VEL
LIN {X 0,Y 319.156,Z 406.626,A -85,B 0,C 180,E1 -18763.483,E2 -18763.483} C_VEL
LIN {X 0,Y 318.632,Z 407.532,A -85,B 0,C 180,E1 -18763.826,E2 -18763.826} C_VEL
LIN {X 0,Y 308.321,Z 422.838,A -85,B 0,C 180,E1 -18765.497,E2 -18765.497} C_VEL
LIN {X 0,Y 298.586,Z 436.747,A -85,B 0,C 180,E1 -18767.412,E2 -18767.412} C_VEL
LIN {X 0,Y 288.619,Z 450.647,A -85,B 0,C 180,E1 -18769.812,E2 -18769.812} C_VEL
LIN {X 0,Y 280.684,Z 461.651,A -85,B 0,C 180,E1 -18772.159,E2 -18772.159} C_VEL
LIN {X 0,Y 272.767,Z 472.751,A -85,B 0,C 180,E1 -18775.019,E2 -18775.019} C_VEL
LIN {X 0,Y 265.873,Z 482.52,A -85,B 0,C 180,E1 -18778.083,E2 -18778.083} C_VEL
LIN {X 0,Y 259.687,Z 491.819,A -85,B 0,C 180,E1 -18781.73,E2 -18781.73} C_VEL
LIN {X 0,Y 254.67,Z 499.656,A -85,B 0,C 180,E1 -18785.546,E2 -18785.546} C_VEL
LIN {X 0,Y 250.997,Z 506.04,A -85,B 0,C 180,E1 -18789.511,E2 -18789.511} C_VEL
LIN {X 0,Y 248.688,Z 510.992,A -85,B 0,C 180,E1 -18793.583,E2 -18793.583} C_VEL
LIN {X 0,Y 247.572,Z 513.843,A -85,B 0,C 180,E1 -18796.872,E2 -18796.872} C_VEL
LIN {X 0,Y 247.102,Z 515.822,A -85,B 0,C 180,E1 -18800.173,E2 -18800.173} C_VEL
LIN {X 0,Y 247.341,Z 516.795,A -85,B 0,C 180,E1 -18803.982,E2 -18803.982} C_VEL
LIN {X 0,Y 247.529,Z 516.66,A -85,B 0,C 180,E1 -18806.744,E2 -18806.744} C_VEL
LIN {X 0,Y 247.988,Z 515.403,A -85,B 0,C 180,E1 -18809.999,E2 -18809.999} C_VEL
LIN {X 0,Y 247.803,Z 512.959,A -85,B 0,C 180,E1 -18813.251,E2 -18813.251} C_VEL
LIN {X 0,Y 247.783,Z 508.629,A -85,B 0,C 180,E1 -18816.919,E2 -18816.919} C_VEL
LIN {X 0,Y 247.671,Z 503.992,A -85,B 0,C 180,E1 -18819.802,E2 -18819.802} C_VEL
LIN {X 0,Y 247.942,Z 497.403,A -85,B 0,C 180,E1 -18823.105,E2 -18823.105} C_VEL
LIN {X 0,Y 248.688,Z 489.215,A -85,B 0,C 180,E1 -18826.414,E2 -18826.414} C_VEL
LIN {X 0,Y 249.947,Z 479.207,A -85,B 0,C 180,E1 -18829.718,E2 -18829.718} C_VEL
LIN {X 0,Y 251.634,Z 468.464,A -85,B 0,C 180,E1 -18832.661,E2 -18832.661} C_VEL
LIN {X 0,Y 253.719,Z 456.464,A -85,B 0,C 180,E1 -18835.425,E2 -18835.425} C_VEL
LIN {X 0,Y 255.954,Z 444.133,A -85,B 0,C 180,E1 -18837.825,E2 -18837.825} C_VEL
LIN {X 0,Y 258.682,Z 429.758,A -85,B 0,C 180,E1 -18840.172,E2 -18840.172} C_VEL
LIN {X 0,Y 261.494,Z 414.109,A -85,B 0,C 180,E1 -18842.286,E2 -18842.286} C_VEL
LIN {X 0,Y 264.295,Z 397.754,A -85,B 0,C 180,E1 -18844.09,E2 -18844.09} C_VEL
LIN {X 0,Y 266.961,Z 380.434,A -85,B 0,C 180,E1 -18845.623,E2 -18845.623} C_VEL
LIN {X 0,Y 269.433,Z 362.257,A -85,B 0,C 180,E1 -18846.864,E2 -18846.864} C_VEL
LIN {X 0,Y 271.198,Z 345.056,A -85,B 0,C 180,E1 -18847.75,E2 -18847.75} C_VEL
LIN {X 0,Y 282.577,Z 206.191,A -85,B 0,C 180,E1 -18853.076,E2 -18853.076} C_VEL
LIN {X 0,Y 282.026,Z 201.903,A -85,B 0,C 180,E1 -18853.336,E2 -18853.336} C_VEL
LIN {X 0,Y 268.752,Z 171.345,A -85,B 0,C 180,E1 -18856.398,E2 -18856.398} C_VEL
LIN {X 0,Y 258.993,Z 150.267,A -85,B 0,C 180,E1 -18858.801,E2 -18858.801} C_VEL
LIN {X 0,Y 253.248,Z 138.189,A -85,B 0,C 180,E1 -18860.336,E2 -18860.336} C_VEL
LIN {X 0,Y 249.054,Z 125.774,A -85,B 0,C 180,E1 -18863.569,E2 -18863.569} C_VEL
LIN {X 0,Y 249.036,Z 125.778,A -85,B 0,C 180,E1 -18867.844,E2 -18867.844} C_VEL
LIN {X 0,Y 249.089,Z 125.77,A -85,B 0,C 180,E1 -18871.338,E2 -18871.338} C_VEL
LIN {X 0,Y 249.147,Z 125.765,A -85,B 0,C 180,E1 -18874.968,E2 -18874.968} C_VEL
LIN {X 0,Y 249.107,Z 125.77,A -85,B 0,C 180,E1 -18880.211,E2 -18880.211} C_VEL
LIN {X 0,Y 249.238,Z 125.749,A -85,B 0,C 180,E1 -18883.622,E2 -18883.622} C_VEL
LIN {X 0,Y 249.249,Z 125.745,A -85,B 0,C 180,E1 -18888.617,E2 -18888.617} C_VEL
LIN {X 0,Y 249.48,Z 125.722,A -85,B 0,C 180,E1 -18891.903,E2 -18891.903} C_VEL
LIN {X 0,Y 249.433,Z 125.722,A -85,B 0,C 180,E1 -18896.77,E2 -18896.77} C_VEL
LIN {X 0,Y 249.731,Z 125.689,A -85,B 0,C 180,E1 -18900,E2 -18900} C_VEL
LIN {X 0,Y 249.433,Z 125.726,A -85,B 0,C 180,E1 -18903.231,E2 -18903.231} C_VEL
LIN {X 0,Y 249.481,Z 125.72,A -85,B 0,C 180,E1 -18908.097,E2 -18908.097} C_VEL
LIN {X 0,Y 249.249,Z 125.748,A -85,B 0,C 180,E1 -18911.384,E2 -18911.384} C_VEL
LIN {X 0,Y 249.238,Z 125.748,A -85,B 0,C 180,E1 -18916.379,E2 -18916.379} C_VEL
LIN {X 0,Y 249.083,Z 125.77,A -85,B 0,C 180,E1 -18921.519,E2 -18921.519} C_VEL
LIN {X 0,Y 249.126,Z 125.765,A -85,B 0,C 180,E1 -18925.482,E2 -18925.482} C_VEL
LIN {X 0,Y 249.079,Z 125.772,A -85,B 0,C 180,E1 -18928.994,E2 -18928.994} C_VEL
LIN {X 0,Y 249.027,Z 125.773,A -85,B 0,C 180,E1 -18932.426,E2 -18932.426} C_VEL
LIN {X 0,Y 249.044,Z 125.774,A -85,B 0,C 180,E1 -18936.343,E2 -18936.343} C_VEL
LIN {X 0,Y 249.003,Z 125.777,A -85,B 0,C 180,E1 -18940.479,E2 -18940.479} C_VEL
LIN {X 0,Y 249.007,Z 125.778,A -85,B 0,C 180,E1 -18944.878,E2 -18944.878} C_VEL
LIN {X 0,Y 249.027,Z 125.773,A -85,B 0,C 180,E1 -18947.367,E2 -18947.367} C_VEL
LIN {X 0,Y 249.049,Z 125.772,A -85,B 0,C 180,E1 -18951.625,E2 -18951.625} C_VEL
LIN {X 0,Y 249.059,Z 125.769,A -85,B 0,C 180,E1 -18955.643,E2 -18955.643} C_VEL
LIN {X 0,Y 249.049,Z 125.772,A -85,B 0,C 180,E1 -18959.474,E2 -18959.474} C_VEL
LIN {X 0,Y 249.071,Z 125.769,A -85,B 0,C 180,E1 -18963.163,E2 -18963.163} C_VEL
LIN {X 0,Y 249.084,Z 125.769,A -85,B 0,C 180,E1 -18966.734,E2 -18966.734} C_VEL
LIN {X 0,Y 249.13,Z 125.762,A -85,B 0,C 180,E1 -18970.214,E2 -18970.214} C_VEL
LIN {X 0,Y 249.242,Z 125.749,A -85,B 0,C 180,E1 -18973.623,E2 -18973.623} C_VEL
LIN {X 0,Y 249.253,Z 125.749,A -85,B 0,C 180,E1 -18978.618,E2 -18978.618} C_VEL
LIN {X 0,Y 249.485,Z 125.717,A -85,B 0,C 180,E1 -18981.904,E2 -18981.904} C_VEL
LIN {X 0,Y 249.437,Z 125.723,A -85,B 0,C 180,E1 -18986.771,E2 -18986.771} C_VEL
LIN {X 0,Y 249.729,Z 125.692,A -85,B 0,C 180,E1 -18990.001,E2 -18990.001} C_VEL
LIN {X 0,Y 249.436,Z 125.717,A -85,B 0,C 180,E1 -18993.231,E2 -18993.231} C_VEL
LIN {X 0,Y 249.486,Z 125.723,A -85,B 0,C 180,E1 -18998.098,E2 -18998.098} C_VEL
LIN {X 0,Y 249.255,Z 125.744,A -85,B 0,C 180,E1 -19001.384,E2 -19001.384} C_VEL
LIN {X 0,Y 249.244,Z 125.749,A -85,B 0,C 180,E1 -19006.379,E2 -19006.379} C_VEL
LIN {X 0,Y 249.091,Z 125.771,A -85,B 0,C 180,E1 -19011.519,E2 -19011.519} C_VEL
LIN {X 0,Y 249.133,Z 125.766,A -85,B 0,C 180,E1 -19015.483,E2 -19015.483} C_VEL
LIN {X 0,Y 249.083,Z 125.771,A -85,B 0,C 180,E1 -19018.993,E2 -19018.993} C_VEL
LIN {X 0,Y 249.039,Z 125.776,A -85,B 0,C 180,E1 -19022.426,E2 -19022.426} C_VEL
